LIN {X 0,Y 254.09,Z 840.895,A -85,B 0,C 180,E1 -18628.414,E2 -18628.414} C_VEL
LIN {X 0,Y 254.062,Z 841.128,A -85,B 0,C 180,E1 -18629.999,E2 -18629.999} C_VEL
LIN {X 0,Y 254.089,Z 840.932,A -85,B 0,C 180,E1 -18631.584,E2 -18631.584} C_VEL
LIN {X 0,Y 254.162,Z 840.345,A -85,B 0,C 180,E1 -18633.169,E2 -18633.169} C_VEL
LIN {X 0,Y 254.513,Z 838.113,A -85,B 0,C 180,E1 -18636.232,E2 -18636.232} C_VEL
LIN {X 0,Y 255.051,Z 835.128,A -85,B 0,C 180,E1 -18638.716,E2 -18638.716} C_VEL
LIN {X 0,Y 255.847,Z 831.213,A -85,B 0,C 180,E1 -18641.085,E2 -18641.085} C_VEL
LIN {X 0,Y 257.022,Z 826.141,A -85,B 0,C 180,E1 -18643.438,E2 -18643.438} C_VEL
LIN {X 0,Y 258.473,Z 819.747,A -85,B 0,C 180,E1 -18645.776,E2 -18645.776} C_VEL
LIN {X 0,Y 260.425,Z 811.783,A -85,B 0,C 180,E1 -18648.078,E2 -18648.078} C_VEL
LIN {X 0,Y 262.234,Z 803.648,A -85,B 0,C 180,E1 -18649.976,E2 -18649.976} C_VEL
LIN {X 0,Y 264.141,Z 793.617,A -85,B 0,C 180,E1 -18651.868,E2 -18651.868} C_VEL
LIN {X 0,Y 266.211,Z 782.348,A -85,B 0,C 180,E1 -18653.533,E2 -18653.533} C_VEL
LIN {X 0,Y 267.959,Z 771.245,A -85,B 0,C 180,E1 -18654.81,E2 -18654.81} C_VEL
LIN {X 0,Y 269.52,Z 758.663,A -85,B 0,C 180,E1 -18655.896,E2 -18655.896} C_VEL
LIN {X 0,Y 270.645,Z 746.284,A -85,B 0,C 180,E1 -18656.662,E2 -18656.662} C_VEL
LIN {X 0,Y 271.369,Z 733.669,A -85,B 0,C 180,E1 -18657.157,E2 -18657.157} C_VEL
LIN {X 0,Y 273.583,Z 662.732,A -85,B 0,C 180,E1 -18658.999,E2 -18658.999} C_VEL
LIN {X 0,Y 269.738,Z 639.631,A -85,B 0,C 180,E1 -18660.151,E2 -18660.151} C_VEL
LIN {X 0,Y 267.312,Z 626.531,A -85,B 0,C 180,E1 -18660.876,E2 -18660.876} C_VEL
LIN {X 0,Y 268.617,Z 614.98,A -85,B 0,C 180,E1 -18663.326,E2 -18663.326} C_VEL
LIN {X 0,Y 267.278,Z 607.072,A -85,B 0,C 180,E1 -18665.399,E2 -18665.399} C_VEL
LIN {X 0,Y 264.897,Z 596.537,A -85,B 0,C 180,E1 -18668.397,E2 -18668.397} C_VEL
LIN {X 0,Y 262.253,Z 586.826,A -85,B 0,C 180,E1 -18671.378,E2 -18671.378} C_VEL
LIN {X 0,Y 261.133,Z 583.175,A -85,B 0,C 180,E1 -18672.573,E2 -18672.573} C_VEL
LIN {X 0,Y 265.751,Z 595.35,A -85,B 0,C 180,E1 -18673.336,E2 -18673.336} C_VEL
LIN {X 0,Y 264.419,Z 646.12,A -85,B 0,C 180,E1 -18675.127,E2 -18675.127} C_VEL
LIN {X 0,Y 264.077,Z 660.633,A -85,B 0,C 180,E1 -18675.846,E2 -18675.846} C_VEL
LIN {X 0,Y 263.423,Z 674.387,A -85,B 0,C 180,E1 -18676.869,E2 -18676.869} C_VEL
LIN {X 0,Y 262.637,Z 685.98,A -85,B 0,C 180,E1 -18678.011,E2 -18678.011} C_VEL
LIN {X 0,Y 261.734,Z 697.28,A -85,B 0,C 180,E1 -18679.417,E2 -18679.417} C_VEL
LIN {X 0,Y 260.579,Z 709.014,A -85,B 0,C 180,E1 -18681.254,E2 -18681.254} C_VEL
LIN {X 0,Y 259.619,Z 718.369,A -85,B 0,C 180,E1 -18683.056,E2 -18683.056} C_VEL
LIN {X 0,Y 258.509,Z 722.566,A -85,B 0,C 180,E1 -18683.944,E2 -18683.944} C_VEL
LIN {X 0,Y 255,Z 729.034,A -85,B 0,C 180,E1 -18685.43,E2 -18685.43} C_VEL
LIN {X 0,Y 251.522,Z 734.947,A -85,B 0,C 180,E1 -18687.059,E2 -18687.059} C_VEL
LIN {X 0,Y 250.487,Z 738.277,A -85,B 0,C 180,E1 -18688.153,E2 -18688.153} C_VEL
LIN {X 0,Y 249.964,Z 744.583,A -85,B 0,C 180,E1 -18690.64,E2 -18690.64} C_VEL
LIN {X 0,Y 249.597,Z 749.74,A -85,B 0,C 180,E1 -18693.223,E2 -18693.223} C_VEL
LIN {X 0,Y 249.477,Z 753.747,A -85,B 0,C 180,E1 -18695.89,E2 -18695.89} C_VEL
LIN {X 0,Y 249.746,Z 756.476,A -85,B 0,C 180,E1 -18698.541,E2 -18698.541} C_VEL
LIN {X 0,Y 250.079,Z 757.631,A -85,B 0,C 180,E1 -18700.291,E2 -18700.291} C_VEL
LIN {X 0,Y 250.675,Z 758.421,A -85,B 0,C 180,E1 -18702.401,E2 -18702.401} C_VEL
LIN {X 0,Y 251.933,Z 758.245,A -85,B 0,C 180,E1 -18705.459,E2 -18705.459} C_VEL
LIN {X 0,Y 252.833,Z 757.518,A -85,B 0,C 180,E1 -18707.151,E2 -18707.151} C_VEL
LIN {X 0,Y 253.866,Z 756.267,A -85,B 0,C 180,E1 -18708.826,E2 -18708.826} C_VEL
LIN {X 0,Y 255.812,Z 753.276,A -85,B 0,C 180,E1 -18711.494,E2 -18711.494} C_VEL
LIN {X 0,Y 257.855,Z 749.625,A -85,B 0,C 180,E1 -18713.741,E2 -18713.741} C_VEL
LIN {X 0,Y 260.549,Z 743.915,A -85,B 0,C 180,E1 -18716.368,E2 -18716.368} C_VEL
LIN {X 0,Y 263.546,Z 736.623,A -85,B 0,C 180,E1 -18718.854,E2 -18718.854} C_VEL
LIN {X 0,Y 266.689,Z 727.942,A -85,B 0,C 180,E1 -18721.171,E2 -18721.171} C_VEL
LIN {X 0,Y 269.312,Z 719.321,A -85,B 0,C 180,E1 -18722.992,E2 -18722.992} C_VEL
LIN {X 0,Y 272.249,Z 708.404,A -85,B 0,C 180,E1 -18724.813,E2 -18724.813} C_VEL
LIN {X 0,Y 274.9,Z 696.038,A -85,B 0,C 180,E1 -18726.422,E2 -18726.422} C_VEL
LIN {X 0,Y 276.654,Z 685.777,A -85,B 0,C 180,E1 -18727.481,E2 -18727.481} C_VEL
LIN {X 0,Y 278.215,Z 673.079,A -85,B 0,C 180,E1 -18728.501,E2 -18728.501} C_VEL
LIN {X 0,Y 279.239,Z 659.814,A -85,B 0,C 180,E1 -18729.262,E2 -18729.262} C_VEL
LIN {X 0,Y 281.024,Z 632.819,A -85,B 0,C 180,E1 -18730.403,E2 -18730.403} C_VEL
LIN {X 0,Y 282.345,Z 617.727,A -85,B 0,C 180,E1 -18730.991,E2 -18730.991} C_VEL
LIN {X 0,Y 278.957,Z 610.736,A -85,B 0,C 180,E1 -18732.326,E2 -18732.326} C_VEL
LIN {X 0,Y 274.251,Z 602.926,A -85,B 0,C 180,E1 -18734.285,E2 -18734.285} C_VEL
LIN {X 0,Y 271.133,Z 598.226,A -85,B 0,C 180,E1 -18735.711,E2 -18735.711} C_VEL
LIN {X 0,Y 269.057,Z 595.035,A -85,B 0,C 180,E1 -18736.773,E2 -18736.773} C_VEL
LIN {X 0,Y 266.386,Z 591.181,A -85,B 0,C 180,E1 -18738.242,E2 -18738.242} C_VEL
LIN {X 0,Y 263.756,Z 587.873,A -85,B 0,C 180,E1 -18739.823,E2 -18739.823} C_VEL
LIN {X 0,Y 263.095,Z 586.506,A -85,B 0,C 180,E1 -18740.32,E2 -18740.32} C_VEL
LIN {X 0,Y 260.443,Z 584.072,A -85,B 0,C 180,E1 -18742.197,E2 -18742.197} C_VEL
LIN {X 0,Y 256.402,Z 580.935,A -85,B 0,C 180,E1 -18746.012,E2 -18746.012} C_VEL
LIN {X 0,Y 253.636,Z 580.564,A -85,B 0,C 180,E1 -18750.802,E2 -18750.802} C_VEL
LIN {X 0,Y 253.372,Z 581.196,A -85,B 0,C 180,E1 -18753.694,E2 -18753.694} C_VEL
LIN {X 0,Y 254.251,Z 583.662,A -85,B 0,C 180,E1 -18756.719,E2 -18756.719} C_VEL
LIN {X 0,Y 255.413,Z 586.748,A -85,B 0,C 180,E1 -18759.543,E2 -18759.543} C_VEL
LIN {X 0,Y 258.229,Z 592.704,A -85,B 0,C 180,E1 -18762.875,E2 -18762.875} C_VEL
LIN {X 0,Y 262.198,Z 599.62,A -85,B 0,C 180,E1 -18766.02,E2 -18766.02} C_VEL
LIN {X 0,Y 266.726,Z 608.628,A -85,B 0,C 180,E1 -18768.878,E2 -18768.878} C_VEL
LIN {X 0,Y 270.377,Z 616.548,A -85,B 0,C 180,E1 -18770.836,E2 -18770.836} C_VEL
LIN {X 0,Y 273.12,Z 623.192,A -85,B 0,C 180,E1 -18772.208,E2 -18772.208} C_VEL
LIN {X 0,Y 274.437,Z 626.568,A -85,B 0,C 180,E1 -18772.82,E2 -18772.82} C_VEL
LIN {X 0,Y 276.106,Z 643.037,A -85,B 0,C 180,E1 -18774.364,E2 -18774.364} C_VEL
LIN {X 0,Y 277.294,Z 660.519,A -85,B 0,C 180,E1 -18775.708,E2 -18775.708} C_VEL
LIN {X 0,Y 277.715,Z 677.5,A -85,B 0,C 180,E1 -18776.784,E2 -18776.784} C_VEL
LIN {X 0,Y 277.476,Z 688.854,A -85,B 0,C 180,E1 -18777.368,E2 -18777.368} C_VEL
LIN {X 0,Y 275.097,Z 715.729,A -85,B 0,C 180,E1 -18778.376,E2 -18778.376} C_VEL
LIN {X 0,Y 273.035,Z 729.581,A -85,B 0,C 180,E1 -18779.125,E2 -18779.125} C_VEL
LIN {X 0,Y 270.167,Z 743.428,A -85,B 0,C 180,E1 -18780.167,E2 -18780.167} C_VEL
LIN {X 0,Y 267.203,Z 755.117,A -85,B 0,C 180,E1 -18781.316,E2 -18781.316} C_VEL
LIN {X 0,Y 263.69,Z 767.153,A -85,B 0,C 180,E1 -18782.845,E2 -18782.845} C_VEL
LIN {X 0,Y 262.11,Z 772.187,A -85,B 0,C 180,E1 -18783.583,E2 -18783.583} C_VEL
LIN {X 0,Y 260.479,Z 784.366,A -85,B 0,C 180,E1 -18784.641,E2 -18784.641} C_VEL
LIN {X 0,Y 258.602,Z 795.598,A -85,B 0,C 180,E1 -18785.944,E2 -18785.944} C_VEL
LIN {X 0,Y 256.382,Z 806.998,A -85,B 0,C 180,E1 -18787.647,E2 -18787.647} C_VEL
LIN {X 0,Y 254.432,Z 816.184,A -85,B 0,C 180,E1 -18789.381,E2 -18789.381} C_VEL
LIN {X 0,Y 252.528,Z 825.133,A -85,B 0,C 180,E1 -18791.5,E2 -18791.5} C_VEL
LIN {X 0,Y 250.784,Z 832.715,A -85,B 0,C 180,E1 -18793.727,E2 -18793.727} C_VEL
LIN {X 0,Y 249.202,Z 839.271,A -85,B 0,C 180,E1 -18796.132,E2 -18796.132} C_VEL
LIN {X 0,Y 248.167,Z 844.485,A -85,B 0,C 180,E1 -18798.568,E2 -18798.568} C_VEL
LIN {X 0,Y 247.485,Z 848.517,A -85,B 0,C 180,E1 -18801.016,E2 -18801.016} C_VEL
LIN {X 0,Y 247.074,Z 851.489,A -85,B 0,C 180,E1 -18803.468,E2 -18803.468} C_VEL
LIN {X 0,Y 246.97,Z 852.915,A -85,B 0,C 180,E1 -18805.104,E2 -18805.104} C_VEL
LIN {X 0,Y 246.977,Z 853.923,A -85,B 0,C 180,E1 -18806.739,E2 -18806.739} C_VEL
LIN {X 0,Y 247.025,Z 854.54,A -85,B 0,C 180,E1 -18808.371,E2 -18808.371} C_VEL
LIN {X 0,Y 247.07,Z 854.757,A -85,B 0,C 180,E1 -18810.001,E2 -18810.001} C_VEL
LIN {X 0,Y 247.015,Z 854.529,A -85,B 0,C 180,E1 -18811.632,E2 -18811.632} C_VEL
LIN {X 0,Y 247.011,Z 852.891,A -85,B 0,C 180,E1 -18814.898,E2 -18814.898} C_VEL
LIN {X 0,Y 247.076,Z 851.449,A -85,B 0,C 180,E1 -18816.534,E2 -18816.534} C_VEL
LIN {X 0,Y 247.508,Z 848.465,A -85,B 0,C 180,E1 -18818.986,E2 -18818.986} C_VEL
LIN {X 0,Y 248.152,Z 844.415,A -85,B 0,C 180,E1 -18821.436,E2 -18821.436} C_VEL
LIN {X 0,Y 249.42,Z 838.173,A -85,B 0,C 180,E1 -18824.275,E2 -18824.275} C_VEL
LIN {X 0,Y 251.04,Z 831.372,A -85,B 0,C 180,E1 -18826.677,E2 -18826.677} C_VEL
LIN {X 0,Y 252.834,Z 823.525,A -85,B 0,C 180,E1 -18828.891,E2 -18828.891} C_VEL
LIN {X 0,Y 254.751,Z 814.094,A -85,B 0,C 180,E1 -18831.018,E2 -18831.018} C_VEL
LIN {X 0,Y 256.841,Z 804.471,A -85,B 0,C 180,E1 -18832.738,E2 -18832.738} C_VEL
LIN {X 0,Y 258.885,Z 793.924,A -85,B 0,C 180,E1 -18834.244,E2 -18834.244} C_VEL
LIN {X 0,Y 260.704,Z 782.098,A -85,B 0,C 180,E1 -18835.553,E2 -18835.553} C_VEL
LIN {X 0,Y 262.332,Z 769.822,A -85,B 0,C 180,E1 -18836.557,E2 -18836.557} C_VEL
LIN {X 0,Y 263.569,Z 758.093,A -85,B 0,C 180,E1 -18837.225,E2 -18837.225} C_VEL
LIN {X 0,Y 264.394,Z 743.701,A -85,B 0,C 180,E1 -18837.723,E2 -18837.723} C_VEL
LIN {X 0,Y 266.125,Z 685.702,A -85,B 0,C 180,E1 -18839.262,E2 -18839.262} C_VEL
LIN {X 0,Y 263.423,Z 657.403,A -85,B 0,C 180,E1 -18840.459,E2 -18840.459} C_VEL
LIN {X 0,Y 260.434,Z 634.29,A -85,B 0,C 180,E1 -18841.594,E2 -18841.594} C_VEL
LIN {X 0,Y 259.764,Z 608.016,A -85,B 0,C 180,E1 -18844.496,E2 -18844.496} C_VEL
LIN {X 0,Y 258.866,Z 603.397,A -85,B 0,C 180,E1 -18845.128,E2 -18845.128} C_VEL
LIN {X 0,Y 254.012,Z 587.934,A -85,B 0,C 180,E1 -18847.655,E2 -18847.655} C_VEL
LIN {X 0,Y 251.33,Z 579.796,A -85,B 0,C 180,E1 -18849.096,E2 -18849.096} C_VEL
LIN {X 0,Y 249.033,Z 569.461,A -85,B 0,C 180,E1 -18852.635,E2 -18852.635} C_VEL
LIN {X 0,Y 249.021,Z 569.455,A -85,B 0,C 180,E1 -18857.364,E2 -18857.364} C_VEL
LIN {X 0,Y 249.046,Z 569.45,A -85,B 0,C 180,E1 -18862.201,E2 -18862.201} C_VEL
LIN {X 0,Y 249.046,Z 569.463,A -85,B 0,C 180,E1 -18865.64,E2 -18865.64} C_VEL
LIN {X 0,Y 249.054,Z 569.44,A -85,B 0,C 180,E1 -18869.473,E2 -18869.473} C_VEL
LIN {X 0,Y 249.073,Z 569.452,A -85,B 0,C 180,E1 -18873.162,E2 -18873.162} C_VEL
LIN {X 0,Y 249.064,Z 569.445,A -85,B 0,C 180,E1 -18876.731,E2 -18876.731} C_VEL
LIN {X 0,Y 249.111,Z 569.443,A -85,B 0,C 180,E1 -18880.212,E2 -18880.212} C_VEL
LIN {X 0,Y 249.226,Z 569.419,A -85,B 0,C 180,E1 -18883.621,E2 -18883.621} C_VEL
LIN {X 0,Y 249.247,Z 569.411,A -85,B 0,C 180,E1 -18888.616,E2 -18888.616} C_VEL
LIN {X 0,Y 249.457,Z 569.401,A -85,B 0,C 180,E1 -18891.902,E2 -18891.902} C_VEL
LIN {X 0,Y 249.297,Z 569.419,A -85,B 0,C 180,E1 -18895.149,E2 -18895.149} C_VEL
LIN {X 0,Y 249.677,Z 569.357,A -85,B 0,C 180,E1 -18898.387,E2 -18898.387} C_VEL
LIN {X 0,Y 249.678,Z 569.384,A -85,B 0,C 180,E1 -18901.613,E2 -18901.613} C_VEL
LIN {X 0,Y 249.451,Z 569.391,A -85,B 0,C 180,E1 -18906.729,E2 -18906.729} C_VEL
LIN {X 0,Y 249.392,Z 569.415,A -85,B 0,C 180,E1 -18909.735,E2 -18909.735} C_VEL
LIN {X 0,Y 249.204,Z 569.436,A -85,B 0,C 180,E1 -18914.704,E2 -18914.704} C_VEL
LIN {X 0,Y 249.142,Z 569.432,A -85,B 0,C 180,E1 -18918.077,E2 -18918.077} C_VEL
LIN {X 0,Y 249.09,Z 569.453,A -85,B 0,C 180,E1 -18921.518,E2 -18921.518} C_VEL
LIN {X 0,Y 249.133,Z 569.43,A -85,B 0,C 180,E1 -18925.482,E2 -18925.482} C_VEL
LIN {X 0,Y 249.086,Z 569.455,A -85,B 0,C 180,E1 -18928.993,E2 -18928.993} C_VEL
LIN {X 0,Y 249.033,Z 569.46,A -85,B 0,C 180,E1 -18932.426,E2 -18932.426} C_VEL
LIN {X 0,Y 249.059,Z 569.453,A -85,B 0,C 180,E1 -18936.341,E2 -18936.341} C_VEL
LIN {X 0,Y 249.029,Z 569.46,A -85,B 0,C 180,E1 -18940.474,E2 -18940.474} C_VEL
LIN {X 0,Y 249.011,Z 569.51,A -85,B 0,C 180,E1 -18943.137,E2 -18943.137} C_VEL
LIN {X 0,Y 253.699,Z 582.025,A -85,B 0,C 180,E1 -18947.232,E2 -18947.232} C_VEL
LIN {X 0,Y 257.124,Z 592.661,A -85,B 0,C 180,E1 -18950.444,E2 -18950.444} C_VEL
LIN {X 0,Y 260.154,Z 603.871,A -85,B 0,C 180,E1 -18953.535,E2 -18953.535} C_VEL
LIN {X 0,Y 262.882,Z 616.414,A -85,B 0,C 180,E1 -18956.711,E2 -18956.711} C_VEL
LIN {X 0,Y 262.799,Z 619.429,A -85,B 0,C 180,E1 -18957.335,E2 -18957.335} C_VEL
LIN {X 0,Y 262.047,Z 625.84,A -85,B 0,C 180,E1 -18958.543,E2 -18958.543} C_VEL
LIN {X 0,Y 266.616,Z 654.96,A -85,B 0,C 180,E1 -18960.056,E2 -18960.056} C_VEL
LIN {X 0,Y 267.466,Z 661.868,A -85,B 0,C 180,E1 -18960.372,E2 -18960.372} C_VEL
LIN {X 0,Y 264.785,Z 738.66,A -85,B 0,C 180,E1 -18962.429,E2 -18962.429} C_VEL
LIN {X 0,Y 263.808,Z 751.811,A -85,B 0,C 180,E1 -18963.07,E2 -18963.07} C_VEL
LIN {X 0,Y 262.417,Z 764.297,A -85,B 0,C 180,E1 -18963.988,E2 -18963.988} C_VEL
LIN {X 0,Y 260.839,Z 775.507,A -85,B 0,C 180,E1 -18965.101,E2 -18965.101} C_VEL
LIN {X 0,Y 258.758,Z 787.098,A -85,B 0,C 180,E1 -18966.594,E2 -18966.594} C_VEL
LIN {X 0,Y 256.708,Z 797.852,A -85,B 0,C 180,E1 -18968.393,E2 -18968.393} C_VEL
LIN {X 0,Y 254.893,Z 806.829,A -85,B 0,C 180,E1 -18970.273,E2 -18970.273} C_VEL
LIN {X 0,Y 252.71,Z 815.756,A -85,B 0,C 180,E1 -18972.604,E2 -18972.604} C_VEL
LIN {X 0,Y 250.925,Z 822.969,A -85,B 0,C 180,E1 -18974.984,E2 -18974.984} C_VEL
LIN {X 0,Y 249.294,Z 829.586,A -85,B 0,C 180,E1 -18977.792,E2 -18977.792} C_VEL
LIN {X 0,Y 248.31,Z 833.924,A -85,B 0,C 180,E1 -18980.221,E2 -18980.221} C_VEL
LIN {X 0,Y 247.845,Z 836.205,A -85,B 0,C 180,E1 -18981.848,E2 -18981.848} C_VEL
LIN {X 0,Y 247.389,Z 838.457,A -85,B 0,C 180,E1 -18983.885,E2 -18983.885} C_VEL
LIN {X 0,Y 247.087,Z 840.476,A -85,B 0,C 180,E1 -18986.738,E2 -18986.738} C_VEL
LIN {X 0,Y 246.992,Z 841.32,A -85,B 0,C 180,E1 -18989.999,E2 -18989.999} C_VEL
LIN {X 0,Y 247,Z 841.125,A -85,B 0,C 180,E1 -18991.629,E2 -18991.629} C_VEL
LIN {X 0,Y 247.084,Z 840.537,A -85,B 0,C 180,E1 -18993.26,E2 -18993.26} C_VEL
LIN {X 0,Y 247.418,Z 838.511,A -85,B 0,C 180,E1 -18996.177,E2 -18996.177} C_VEL
LIN {X 0,Y 248.042,Z 835.319,A -85,B 0,C 180,E1 -18998.964,E2 -18998.964} C_VEL
LIN {X 0,Y 248.875,Z 831.404,A -85,B 0,C 180,E1 -19001.399,E2 -19001.399} C_VEL
LIN {X 0,Y 250.114,Z 826.331,A -85,B 0,C 180,E1 -19003.817,E2 -19003.817} C_VEL
LIN {X 0,Y 251.642,Z 819.935,A -85,B 0,C 180,E1 -19006.216,E2 -19006.216} C_VEL
LIN {X 0,Y 253.691,Z 811.969,A -85,B 0,C 180,E1 -19008.576,E2 -19008.576} C_VEL
LIN {X 0,Y 255.675,Z 803.234,A -85,B 0,C 180,E1 -19010.653,E2 -19010.653} C_VEL
LIN {X 0,Y 257.574,Z 793.796,A -85,B 0,C 180,E1 -19012.456,E2 -19012.456} C_VEL
LIN {X 0,Y 259.738,Z 782.522,A -85,B 0,C 180,E1 -19014.156,E2 -19014.156} C_VEL
LIN {X 0,Y 261.545,Z 771.411,A -85,B 0,C 180,E1 -19015.462,E2 -19015.462} C_VEL
LIN {X 0,Y 263.034,Z 760.044,A -85,B 0,C 180,E1 -19016.477,E2 -19016.477} C_VEL
LIN {X 0,Y 264.257,Z 747.263,A -85,B 0,C 180,E1 -19017.306,E2 -19017.306} C_VEL
LIN {X 0,Y 265.04,Z 735.241,A -85,B 0,C 180,E1 -19017.807,E2 -19017.807} C_VEL
LIN {X 0,Y 267.411,Z 663.775,A -85,B 0,C 180,E1 -19019.704,E2 -19019.704} C_VEL
LIN {X 0,Y 263.005,Z 637.473,A -85,B 0,C 180,E1 -19021.076,E2 -19021.076} C_VEL
LIN {X 0,Y 261,Z 626.634,A -85,B 0,C 180,E1 -19021.701,E2 -19021.701} C_VEL
LIN {X 0,Y 262.114,Z 617.018,A -85,B 0,C 180,E1 -19023.778,E2 -19023.778} C_VEL
LIN {X 0,Y 260.389,Z 607.236,A -85,B 0,C 180,E1 -19026.424,E2 -19026.424} C_VEL
LIN {X 0,Y 257.403,Z 594.767,A -85,B 0,C 180,E1 -19030.137,E2 -19030.137} C_VEL
LIN {X 0,Y 255.388,Z 587.888,A -85,B 0,C 180,E1 -19032.362,E2 -19032.362} C_VEL
LIN {X 0,Y 256.803,Z 590.995,A -85,B 0,C 180,E1 -19032.577,E2 -19032.577} C_VEL
LIN {X 0,Y 259.068,Z 597.539,A -85,B 0,C 180,E1 -19032.98,E2 -19032.98} C_VEL
LIN {X 0,Y 257.655,Z 639.19,A -85,B 0,C 180,E1 -19034.476,E2 -19034.476} C_VEL
LIN {X 0,Y 257.372,Z 656.39,A -85,B 0,C 180,E1 -19035.21,E2 -19035.21} C_VEL
LIN {X 0,Y 256.764,Z 670.302,A -85,B 0,C 180,E1 -19036.144,E2 -19036.144} C_VEL
LIN {X 0,Y 256.037,Z 682.338,A -85,B 0,C 180,E1 -19037.244,E2 -19037.244} C_VEL
LIN {X 0,Y 255.137,Z 694.009,A -85,B 0,C 180,E1 -19038.616,E2 -19038.616} C_VEL
LIN {X 0,Y 253.941,Z 706.445,A -85,B 0,C 180,E1 -19040.465,E2 -19040.465} C_VEL
LIN {X 0,Y 252.919,Z 716.407,A -85,B 0,C 180,E1 -19042.314,E2 -19042.314} C_VEL
LIN {X 0,Y 251.822,Z 726.426,A -85,B 0,C 180,E1 -19044.612,E2 -19044.612} C_VEL
LIN {X 0,Y 250.987,Z 733.793,A -85,B 0,C 180,E1 -19046.675,E2 -19046.675} C_VEL
LIN {X 0,Y 250.487,Z 738.277,A -85,B 0,C 180,E1 -19048.153,E2 -19048.153} C_VEL
LIN {X 0,Y 249.499,Z 741.431,A -85,B 0,C 180,E1 -19049.279,E2 -19049.279} C_VEL
LIN {X 0,Y 246.27,Z 746.193,A -85,B 0,C 180,E1 -19051.148,E2 -19051.148} C_VEL
LIN {X 0,Y 243.18,Z 750.314,A -85,B 0,C 180,E1 -19053.139,E2 -19053.139} C_VEL
LIN {X 0,Y 242.435,Z 752.446,A -85,B 0,C 180,E1 -19054.432,E2 -19054.432} C_VEL
LIN {X 0,Y 242.422,Z 754.701,A -85,B 0,C 180,E1 -19056.054,E2 -19056.054} C_VEL
LIN {X 0,Y 242.601,Z 756.771,A -85,B 0,C 180,E1 -19057.969,E2 -19057.969} C_VEL
LIN {X 0,Y 242.91,Z 758.159,A -85,B 0,C 180,E1 -19059.684,E2 -19059.684} C_VEL
LIN {X 0,Y 243.577,Z 759.382,A -85,B 0,C 180,E1 -19062.198,E2 -19062.198} C_VEL
LIN {X 0,Y 244.686,Z 759.623,A -85,B 0,C 180,E1 -19065.019,E2 -19065.019} C_VEL
LIN {X 0,Y 245.597,Z 759.147,A -85,B 0,C 180,E1 -19066.766,E2 -19066.766} C_VEL
LIN {X 0,Y 246.642,Z 758.193,A -85,B 0,C 180,E1 -19068.494,E2 -19068.494} C_VEL
LIN {X 0,Y 248.753,Z 755.486,A -85,B 0,C 180,E1 -19071.422,E2 -19071.422} C_VEL
LIN {X 0,Y 250.65,Z 752.454,A -85,B 0,C 180,E1 -19073.56,E2 -19073.56} C_VEL
LIN {X 0,Y 253.518,Z 747.121,A -85,B 0,C 180,E1 -19076.329,E2 -19076.329} C_VEL
LIN {X 0,Y 256.507,Z 740.69,A -85,B 0,C 180,E1 -19078.822,E2 -19078.822} C_VEL
LIN {X 0,Y 259.282,Z 733.984,A -85,B 0,C 180,E1 -19080.854,E2 -19080.854} C_VEL
LIN {X 0,Y 262.174,Z 725.886,A -85,B 0,C 180,E1 -19082.839,E2 -19082.839} C_VEL
LIN {X 0,Y 265.177,Z 716.123,A -85,B 0,C 180,E1 -19084.751,E2 -19084.751} C_VEL
LIN {X 0,Y 268.104,Z 705.231,A -85,B 0,C 180,E1 -19086.434,E2 -19086.434} C_VEL
LIN {X 0,Y 270.598,Z 693.198,A -85,B 0,C 180,E1 -19087.894,E2 -19087.894} C_VEL
LIN {X 0,Y 272.646,Z 680.632,A -85,B 0,C 180,E1 -19089.053,E2 -19089.053} C_VEL
LIN {X 0,Y 274.025,Z 667.183,A -85,B 0,C 180,E1 -19089.999,E2 -19089.999} C_VEL
LIN {X 0,Y 275.305,Z 648.329,A -85,B 0,C 180,E1 -19090.905,E2 -19090.905} C_VEL
LIN {X 0,Y 277.684,Z 620.883,A -85,B 0,C 180,E1 -19092.021,E2 -19092.021} C_VEL
LIN {X 0,Y 275.405,Z 615.981,A -85,B 0,C 180,E1 -19092.991,E2 -19092.991} C_VEL
LIN {X 0,Y 270.894,Z 608.299,A -85,B 0,C 180,E1 -19094.985,E2 -19094.985} C_VEL
LIN {X 0,Y 266.537,Z 601.354,A -85,B 0,C 180,E1 -19097.216,E2 -19097.216} C_VEL
LIN {X 0,Y 263.964,Z 597.532,A -85,B 0,C 180,E1 -19098.733,E2 -19098.733} C_VEL
LIN {X 0,Y 261.41,Z 594.02,A -85,B 0,C 180,E1 -19100.39,E2 -19100.39} C_VEL
LIN {X 0,Y 260.837,Z 593.011,A -85,B 0,C 180,E1 -19100.839,E2 -19100.839} C_VEL
LIN {X 0,Y 258.203,Z 590.417,A -85,B 0,C 180,E1 -19102.822,E2 -19102.822} C_VEL
LIN {X 0,Y 255.21,Z 588.146,A -85,B 0,C 180,E1 -19105.729,E2 -19105.729} C_VEL
LIN {X 0,Y 253.396,Z 587.616,A -85,B 0,C 180,E1 -19108.132,E2 -19108.132} C_VEL
LIN {X 0,Y 252.16,Z 587.56,A -85,B 0,C 180,E1 -19111.129,E2 -19111.129} C_VEL
LIN {X 0,Y 251.929,Z 588.384,A -85,B 0,C 180,E1 -19113.913,E2 -19113.913} C_VEL
LIN {X 0,Y 252.608,Z 590.937,A -85,B 0,C 180,E1 -19116.996,E2 -19116.996} C_VEL
LIN {X 0,Y 253.732,Z 593.511,A -85,B 0,C 180,E1 -19119.214,E2 -19119.214} C_VEL
LIN {X 0,Y 256.46,Z 599.656,A -85,B 0,C 180,E1 -19122.636,E2 -19122.636} C_VEL
LIN {X 0,Y 259.717,Z 605.662,A -85,B 0,C 180,E1 -19125.384,E2 -19125.384} C_VEL
LIN {X 0,Y 263.844,Z 614.341,A -85,B 0,C 180,E1 -19128.195,E2 -19128.195} C_VEL
LIN {X 0,Y 267.113,Z 621.867,A -85,B 0,C 180,E1 -19130.108,E2 -19130.108} C_VEL
LIN {X 0,Y 269.665,Z 628.359,A -85,B 0,C 180,E1 -19131.477,E2 -19131.477} C_VEL
LIN {X 0,Y 270.426,Z 630.865,A -85,B 0,C 180,E1 -19131.914,E2 -19131.914} C_VEL
LIN {X 0,Y 271.947,Z 648.046,A -85,B 0,C 180,E1 -19133.533,E2 -19133.533} C_VEL
LIN {X 0,Y 272.788,Z 665.923,A -85,B 0,C 180,E1 -19134.925,E2 -19134.925} C_VEL
LIN {X 0,Y 272.877,Z 684.026,A -85,B 0,C 180,E1 -19136.018,E2 -19136.018} C_VEL
LIN {X 0,Y 272.525,Z 691.059,A -85,B 0,C 180,E1 -19136.346,E2 -19136.346} C_VEL
LIN {X 0,Y 270.201,Z 714.937,A -85,B 0,C 180,E1 -19137.283,E2 -19137.283} C_VEL
LIN {X 0,Y 268.004,Z 728.536,A -85,B 0,C 180,E1 -19138.038,E2 -19138.038} C_VEL
LIN {X 0,Y 265,Z 742.273,A -85,B 0,C 180,E1 -19139.082,E2 -19139.082} C_VEL
LIN {X 0,Y 261.917,Z 753.948,A -85,B 0,C 180,E1 -19140.239,E2 -19140.239} C_VEL
LIN {X 0,Y 258.233,Z 765.958,A -85,B 0,C 180,E1 -19141.781,E2 -19141.781} C_VEL
LIN {X 0,Y 255.527,Z 773.89,A -85,B 0,C 180,E1 -19143.013,E2 -19143.013} C_VEL
LIN {X 0,Y 253.804,Z 785.941,A -85,B 0,C 180,E1 -19144.145,E2 -19144.145} C_VEL
LIN {X 0,Y 251.864,Z 796.83,A -85,B 0,C 180,E1 -19145.478,E2 -19145.478} C_VEL
LIN {X 0,Y 249.568,Z 807.936,A -85,B 0,C 180,E1 -19147.221,E2 -19147.221} C_VEL
LIN {X 0,Y 247.366,Z 817.776,A -85,B 0,C 180,E1 -19149.2,E2 -19149.2} C_VEL
LIN {X 0,Y 245.619,Z 825.59,A -85,B 0,C 180,E1 -19151.149,E2 -19151.149} C_VEL
LIN {X 0,Y 243.665,Z 833.749,A -85,B 0,C 180,E1 -19153.669,E2 -19153.669} C_VEL
LIN {X 0,Y 242.287,Z 839.081,A -85,B 0,C 180,E1 -19155.728,E2 -19155.728} C_VEL
LIN {X 0,Y 241.187,Z 844.293,A -85,B 0,C 180,E1 -19158.232,E2 -19158.232} C_VEL
LIN {X 0,Y 240.44,Z 848.325,A -85,B 0,C 180,E1 -19160.75,E2 -19160.75} C_VEL
LIN {X 0,Y 239.997,Z 851.296,A -85,B 0,C 180,E1 -19163.275,E2 -19163.275} C_VEL
LIN {X 0,Y 239.88,Z 852.722,A -85,B 0,C 180,E1 -19164.959,E2 -19164.959} C_VEL
LIN {X 0,Y 239.877,Z 853.73,A -85,B 0,C 180,E1 -19166.642,E2 -19166.642} C_VEL
LIN {X 0,Y 239.931,Z 854.347,A -85,B 0,C 180,E1 -19168.323,E2 -19168.323} C_VEL
LIN {X 0,Y 239.997,Z 854.565,A -85,B 0,C 180,E1 -19170.001,E2 -19170.001} C_VEL
LIN {X 0,Y 239.922,Z 854.336,A -85,B 0,C 180,E1 -19171.68,E2 -19171.68} C_VEL
LIN {X 0,Y 239.921,Z 852.697,A -85,B 0,C 180,E1 -19175.043,E2 -19175.043} C_VEL
LIN {X 0,Y 240.001,Z 851.255,A -85,B 0,C 180,E1 -19176.728,E2 -19176.728} C_VEL
LIN {X 0,Y 240.456,Z 848.27,A -85,B 0,C 180,E1 -19179.252,E2 -19179.252} C_VEL
LIN {X 0,Y 241.166,Z 844.221,A -85,B 0,C 180,E1 -19181.772,E2 -19181.772} C_VEL
LIN {X 0,Y 242.529,Z 837.98,A -85,B 0,C 180,E1 -19184.689,E2 -19184.689} C_VEL
LIN {X 0,Y 244.182,Z 831.178,A -85,B 0,C 180,E1 -19187.16,E2 -19187.16} C_VEL
LIN {X 0,Y 245.941,Z 824.007,A -85,B 0,C 180,E1 -19189.252,E2 -19189.252} C_VEL
LIN {X 0,Y 247.699,Z 815.836,A -85,B 0,C 180,E1 -19191.209,E2 -19191.209} C_VEL
LIN {X 0,Y 250.035,Z 805.446,A -85,B 0,C 180,E1 -19193.174,E2 -19193.174} C_VEL
LIN {X 0,Y 252.129,Z 795.159,A -85,B 0,C 180,E1 -19194.717,E2 -19194.717} C_VEL
LIN {X 0,Y 254.048,Z 783.861,A -85,B 0,C 180,E1 -19196.052,E2 -19196.052} C_VEL
LIN {X 0,Y 255.847,Z 770.923,A -85,B 0,C 180,E1 -19197.174,E2 -19197.174} C_VEL
LIN {X 0,Y 257.188,Z 758.88,A -85,B 0,C 180,E1 -19197.9,E2 -19197.9} C_VEL
LIN {X 0,Y 258.06,Z 745.717,A -85,B 0,C 180,E1 -19198.396,E2 -19198.396} C_VEL
LIN {X 0,Y 259.901,Z 685.945,A -85,B 0,C 180,E1 -19200.023,E2 -19200.023} C_VEL
LIN {X 0,Y 257.251,Z 657.764,A -85,B 0,C 180,E1 -19201.257,E2 -19201.257} C_VEL
LIN {X 0,Y 254.175,Z 634.196,A -85,B 0,C 180,E1 -19202.469,E2 -19202.469} C_VEL
LIN {X 0,Y 253.843,Z 610.077,A -85,B 0,C 180,E1 -19205.241,E2 -19205.241} C_VEL
LIN {X 0,Y 252.81,Z 605.724,A -85,B 0,C 180,E1 -19205.882,E2 -19205.882} C_VEL
LIN {X 0,Y 249.822,Z 596.027,A -85,B 0,C 180,E1 -19207.512,E2 -19207.512} C_VEL
LIN {X 0,Y 245.651,Z 582.707,A -85,B 0,C 180,E1 -19209.925,E2 -19209.925} C_VEL
LIN {X 0,Y 242.755,Z 573.824,A -85,B 0,C 180,E1 -19211.75,E2 -19211.75} C_VEL
LIN {X 0,Y 241.964,Z 570.336,A -85,B 0,C 180,E1 -19213.076,E2 -19213.076} C_VEL
LIN {X 0,Y 241.939,Z 570.346,A -85,B 0,C 180,E1 -19216.571,E2 -19216.571} C_VEL
LIN {X 0,Y 241.959,Z 570.345,A -85,B 0,C 180,E1 -19220.281,E2 -19220.281} C_VEL
LIN {X 0,Y 241.983,Z 570.329,A -85,B 0,C 180,E1 -19224.488,E2 -19224.488} C_VEL
LIN {X 0,Y 241.977,Z 570.321,A -85,B 0,C 180,E1 -19228.48,E2 -19228.48} C_VEL
LIN {X 0,Y 242.01,Z 570.339,A -85,B 0,C 180,E1 -19232.313,E2 -19232.313} C_VEL
LIN {X 0,Y 242.044,Z 570.311,A -85,B 0,C 180,E1 -19236.015,E2 -19236.015} C_VEL
LIN {X 0,Y 242.038,Z 570.331,A -85,B 0,C 180,E1 -19239.608,E2 -19239.608} C_VEL
LIN {X 0,Y 242.166,Z 570.294,A -85,B 0,C 180,E1 -19243.278,E2 -19243.278} C_VEL
LIN {X 0,Y 242.183,Z 570.294,A -85,B 0,C 180,E1 -19248.28,E2 -19248.28} C_VEL
LIN {X 0,Y 242.403,Z 570.276,A -85,B 0,C 180,E1 -19251.665,E2 -19251.665} C_VEL
LIN {X 0,Y 242.258,Z 570.297,A -85,B 0,C 180,E1 -19255.007,E2 -19255.007} C_VEL
LIN {X 0,Y 242.638,Z 570.232,A -85,B 0,C 180,E1 -19258.34,E2 -19258.34} C_VEL
LIN {X 0,Y 242.638,Z 570.261,A -85,B 0,C 180,E1 -19261.66,E2 -19261.66} C_VEL
LIN {X 0,Y 242.431,Z 570.266,A -85,B 0,C 180,E1 -19266.706,E2 -19266.706} C_VEL
LIN {X 0,Y 242.317,Z 570.294,A -85,B 0,C 180,E1 -19270.022,E2 -19270.022} C_VEL
LIN {X 0,Y 242.167,Z 570.317,A -85,B 0,C 180,E1 -19275.141,E2 -19275.141} C_VEL
LIN {X 0,Y 242.075,Z 570.307,A -85,B 0,C 180,E1 -19278.624,E2 -19278.624} C_VEL
LIN {X 0,Y 242.016,Z 570.34,A -85,B 0,C 180,E1 -19282.18,E2 -19282.18} C_VEL
LIN {X 0,Y 242.07,Z 570.311,A -85,B 0,C 180,E1 -19285.838,E2 -19285.838} C_VEL
LIN {X 0,Y 242.033,Z 570.325,A -85,B 0,C 180,E1 -19289.58,E2 -19289.58} C_VEL
LIN {X 0,Y 241.985,Z 570.346,A -85,B 0,C 180,E1 -19293.492,E2 -19293.492} C_VEL
LIN {X 0,Y 242.002,Z 570.345,A -85,B 0,C 180,E1 -19297.58,E2 -19297.58} C_VEL
LIN {X 0,Y 241.943,Z 570.406,A -85,B 0,C 180,E1 -19301.714,E2 -19301.714} C_VEL
LIN {X 0,Y 246.074,Z 581.311,A -85,B 0,C 180,E1 -19305.563,E2 -19305.563} C_VEL
LIN {X 0,Y 249.569,Z 591.221,A -85,B 0,C 180,E1 -19308.705,E2 -19308.705} C_VEL
LIN {X 0,Y 252.451,Z 601.155,A -85,B 0,C 180,E1 -19311.643,E2 -19311.643} C_VEL
LIN {X 0,Y 255.514,Z 614.014,A -85,B 0,C 180,E1 -19315.069,E2 -19315.069} C_VEL
LIN {X 0,Y 256.572,Z 619.642,A -85,B 0,C 180,E1 -19316.465,E2 -19316.465} C_VEL
LIN {X 0,Y 255.815,Z 626,A -85,B 0,C 180,E1 -19317.697,E2 -19317.697} C_VEL
LIN {X 0,Y 260.073,Z 653.291,A -85,B 0,C 180,E1 -19319.166,E2 -19319.166} C_VEL
LIN {X 0,Y 261.288,Z 663.431,A -85,B 0,C 180,E1 -19319.645,E2 -19319.645} C_VEL
LIN {X 0,Y 258.529,Z 738.791,A -85,B 0,C 180,E1 -19321.703,E2 -19321.703} C_VEL
LIN {X 0,Y 257.518,Z 751.975,A -85,B 0,C 180,E1 -19322.357,E2 -19322.357} C_VEL
LIN {X 0,Y 256.073,Z 764.47,A -85,B 0,C 180,E1 -19323.293,E2 -19323.293} C_VEL
LIN {X 0,Y 254.434,Z 775.687,A -85,B 0,C 180,E1 -19324.43,E2 -19324.43} C_VEL
LIN {X 0,Y 252.256,Z 787.284,A -85,B 0,C 180,E1 -19325.954,E2 -19325.954} C_VEL
LIN {X 0,Y 250.111,Z 798.041,A -85,B 0,C 180,E1 -19327.793,E2 -19327.793} C_VEL
LIN {X 0,Y 248.187,Z 807.16,A -85,B 0,C 180,E1 -19329.752,E2 -19329.752} C_VEL
LIN {X 0,Y 245.954,Z 815.947,A -85,B 0,C 180,E1 -19332.11,E2 -19332.11} C_VEL
LIN {X 0,Y 244.07,Z 823.162,A -85,B 0,C 180,E1 -19334.551,E2 -19334.551} C_VEL
LIN {X 0,Y 242.342,Z 829.78,A -85,B 0,C 180,E1 -19337.436,E2 -19337.436} C_VEL
LIN {X 0,Y 241.304,Z 834.118,A -85,B 0,C 180,E1 -19339.935,E2 -19339.935} C_VEL
LIN {X 0,Y 240.807,Z 836.398,A -85,B 0,C 180,E1 -19341.608,E2 -19341.608} C_VEL
LIN {X 0,Y 240.304,Z 838.834,A -85,B 0,C 180,E1 -19343.923,E2 -19343.923} C_VEL
LIN {X 0,Y 240.01,Z 840.669,A -85,B 0,C 180,E1 -19346.641,E2 -19346.641} C_VEL
LIN {X 0,Y 239.923,Z 841.512,A -85,B 0,C 180,E1 -19349.999,E2 -19349.999} C_VEL
LIN {X 0,Y 239.912,Z 841.317,A -85,B 0,C 180,E1 -19351.677,E2 -19351.677} C_VEL
LIN {X 0,Y 240.008,Z 840.729,A -85,B 0,C 180,E1 -19353.356,E2 -19353.356} C_VEL
LIN {X 0,Y 240.318,Z 838.914,A -85,B 0,C 180,E1 -19356.109,E2 -19356.109} C_VEL
LIN {X 0,Y 241.011,Z 835.511,A -85,B 0,C 180,E1 -19359.228,E2 -19359.228} C_VEL
LIN {X 0,Y 241.916,Z 831.595,A -85,B 0,C 180,E1 -19361.732,E2 -19361.732} C_VEL
LIN {X 0,Y 243.219,Z 826.52,A -85,B 0,C 180,E1 -19364.216,E2 -19364.216} C_VEL
LIN {X 0,Y 244.83,Z 820.123,A -85,B 0,C 180,E1 -19366.68,E2 -19366.68} C_VEL
LIN {X 0,Y 246.979,Z 812.154,A -85,B 0,C 180,E1 -19369.1,E2 -19369.1} C_VEL
LIN {X 0,Y 248.908,Z 803.975,A -85,B 0,C 180,E1 -19371.106,E2 -19371.106} C_VEL
LIN {X 0,Y 251.034,Z 793.976,A -85,B 0,C 180,E1 -19373.074,E2 -19373.074} C_VEL
LIN {X 0,Y 253.288,Z 782.696,A -85,B 0,C 180,E1 -19374.812,E2 -19374.812} C_VEL
LIN {X 0,Y 255.161,Z 771.578,A -85,B 0,C 180,E1 -19376.146,E2 -19376.146} C_VEL
LIN {X 0,Y 256.843,Z 758.97,A -85,B 0,C 180,E1 -19377.277,E2 -19377.277} C_VEL
LIN {X 0,Y 258.069,Z 746.551,A -85,B 0,C 180,E1 -19378.073,E2 -19378.073} C_VEL
LIN {X 0,Y 258.862,Z 733.81,A -85,B 0,C 180,E1 -19378.586,E2 -19378.586} C_VEL
LIN {X 0,Y 261.202,Z 664.421,A -85,B 0,C 180,E1 -19380.466,E2 -19380.466} C_VEL
LIN {X 0,Y 256.549,Z 636.372,A -85,B 0,C 180,E1 -19381.987,E2 -19381.987} C_VEL
LIN {X 0,Y 254.753,Z 626.786,A -85,B 0,C 180,E1 -19382.579,E2 -19382.579} C_VEL
LIN {X 0,Y 255.597,Z 618.433,A -85,B 0,C 180,E1 -19384.422,E2 -19384.422} C_VEL
LIN {X 0,Y 253.4,Z 607.174,A -85,B 0,C 180,E1 -19387.599,E2 -19387.599} C_VEL
LIN {X 0,Y 250.842,Z 596.665,A -85,B 0,C 180,E1 -19390.845,E2 -19390.845} C_VEL
LIN {X 0,Y 249.715,Z 592.683,A -85,B 0,C 180,E1 -19392.171,E2 -19392.171} C_VEL
LIN {X 0,Y 251.194,Z 595.873,A -85,B 0,C 180,E1 -19392.398,E2 -19392.398} C_VEL
LIN {X 0,Y 252.164,Z 599.245,A -85,B 0,C 180,E1 -19392.596,E2 -19392.596} C_VEL
LIN {X 0,Y 250.725,Z 641.596,A -85,B 0,C 180,E1 -19394.176,E2 -19394.176} C_VEL
LIN {X 0,Y 250.442,Z 657.573,A -85,B 0,C 180,E1 -19394.891,E2 -19394.891} C_VEL
LIN {X 0,Y 249.858,Z 670.554,A -85,B 0,C 180,E1 -19395.781,E2 -19395.781} C_VEL
LIN {X 0,Y 249.055,Z 683.719,A -85,B 0,C 180,E1 -19397.011,E2 -19397.011} C_VEL
LIN {X 0,Y 248.015,Z 696.014,A -85,B 0,C 180,E1 -19398.518,E2 -19398.518} C_VEL
LIN {X 0,Y 246.972,Z 706.977,A -85,B 0,C 180,E1 -19400.201,E2 -19400.201} C_VEL
LIN {X 0,Y 245.901,Z 716.993,A -85,B 0,C 180,E1 -19402.085,E2 -19402.085} C_VEL
LIN {X 0,Y 244.795,Z 727.117,A -85,B 0,C 180,E1 -19404.453,E2 -19404.453} C_VEL
LIN {X 0,Y 243.817,Z 735.271,A -85,B 0,C 180,E1 -19406.792,E2 -19406.792} C_VEL
LIN {X 0,Y 243.123,Z 742.781,A -85,B 0,C 180,E1 -19409.505,E2 -19409.505} C_VEL
LIN {X 0,Y 242.633,Z 749.017,A -85,B 0,C 180,E1 -19412.39,E2 -19412.39} C_VEL
LIN {X 0,Y 242.435,Z 752.446,A -85,B 0,C 180,E1 -19414.432,E2 -19414.432} C_VEL
LIN {X 0,Y 241.758,Z 754.381,A -85,B 0,C 180,E1 -19415.746,E2 -19415.746} C_VEL
LIN {X 0,Y 239.078,Z 757.134,A -85,B 0,C 180,E1 -19417.924,E2 -19417.924} C_VEL
LIN {X 0,Y 236.985,Z 758.9,A -85,B 0,C 180,E1 -19419.724,E2 -19419.724} C_VEL
LIN {X 0,Y 236.298,Z 759.884,A -85,B 0,C 180,E1 -19421.13,E2 -19421.13} C_VEL
LIN {X 0,Y 236.352,Z 760.115,A -85,B 0,C 180,E1 -19421.604,E2 -19421.604} C_VEL
LIN {X 0,Y 237.445,Z 760.847,A -85,B 0,C 180,E1 -19424.55,E2 -19424.55} C_VEL
LIN {X 0,Y 238.446,Z 760.579,A -85,B 0,C 180,E1 -19426.559,E2 -19426.559} C_VEL
LIN {X 0,Y 239.393,Z 759.977,A -85,B 0,C 180,E1 -19428.141,E2 -19428.141} C_VEL
LIN {X 0,Y 240.577,Z 758.849,A -85,B 0,C 180,E1 -19429.905,E2 -19429.905} C_VEL
LIN {X 0,Y 242.64,Z 756.242,A -85,B 0,C 180,E1 -19432.511,E2 -19432.511} C_VEL
LIN {X 0,Y 245.141,Z 752.486,A -85,B 0,C 180,E1 -19435.066,E2 -19435.066} C_VEL
LIN {X 0,Y 247.898,Z 747.526,A -85,B 0,C 180,E1 -19437.563,E2 -19437.563} C_VEL
LIN {X 0,Y 251.062,Z 741.134,A -85,B 0,C 180,E1 -19440,E2 -19440} C_VEL
LIN {X 0,Y 254.423,Z 733.327,A -85,B 0,C 180,E1 -19442.314,E2 -19442.314} C_VEL
LIN {X 0,Y 257.461,Z 724.991,A -85,B 0,C 180,E1 -19444.305,E2 -19444.305} C_VEL
LIN {X 0,Y 260.396,Z 716.03,A -85,B 0,C 180,E1 -19446.003,E2 -19446.003} C_VEL
LIN {X 0,Y 262.921,Z 706.924,A -85,B 0,C 180,E1 -19447.411,E2 -19447.411} C_VEL
LIN {X 0,Y 265.555,Z 695.346,A -85,B 0,C 180,E1 -19448.864,E2 -19448.864} C_VEL
LIN {X 0,Y 267.69,Z 683.478,A -85,B 0,C 180,E1 -19450.017,E2 -19450.017} C_VEL
LIN {X 0,Y 269.245,Z 670.621,A -85,B 0,C 180,E1 -19450.973,E2 -19450.973} C_VEL
LIN {X 0,Y 270.592,Z 652.317,A -85,B 0,C 180,E1 -19451.908,E2 -19451.908} C_VEL
LIN {X 0,Y 273.175,Z 623.823,A -85,B 0,C 180,E1 -19453.118,E2 -19453.118} C_VEL
LIN {X 0,Y 269.754,Z 617.274,A -85,B 0,C 180,E1 -19454.682,E2 -19454.682} C_VEL
LIN {X 0,Y 265.449,Z 609.996,A -85,B 0,C 180,E1 -19456.885,E2 -19456.885} C_VEL
LIN {X 0,Y 263.21,Z 606.44,A -85,B 0,C 180,E1 -19458.185,E2 -19458.185} C_VEL
LIN {X 0,Y 261.506,Z 603.768,A -85,B 0,C 180,E1 -19459.267,E2 -19459.267} C_VEL
LIN {X 0,Y 259.065,Z 600.14,A -85,B 0,C 180,E1 -19461,E2 -19461} C_VEL
LIN {X 0,Y 257.726,Z 598.663,A -85,B 0,C 180,E1 -19462.01,E2 -19462.01} C_VEL
LIN {X 0,Y 256.477,Z 597.222,A -85,B 0,C 180,E1 -19463.074,E2 -19463.074} C_VEL
LIN {X 0,Y 253.712,Z 595.068,A -85,B 0,C 180,E1 -19465.845,E2 -19465.845} C_VEL
LIN {X 0,Y 251.897,Z 594.554,A -85,B 0,C 180,E1 -19468.314,E2 -19468.314} C_VEL
LIN {X 0,Y 250.738,Z 594.565,A -85,B 0,C 180,E1 -19471.326,E2 -19471.326} C_VEL
LIN {X 0,Y 250.529,Z 595.334,A -85,B 0,C 180,E1 -19473.776,E2 -19473.776} C_VEL
LIN {X 0,Y 251.077,Z 597.747,A -85,B 0,C 180,E1 -19476.701,E2 -19476.701} C_VEL
LIN {X 0,Y 252.055,Z 600.21,A -85,B 0,C 180,E1 -19478.832,E2 -19478.832} C_VEL
LIN {X 0,Y 254.671,Z 606.524,A -85,B 0,C 180,E1 -19482.36,E2 -19482.36} C_VEL
LIN {X 0,Y 257.306,Z 611.696,A -85,B 0,C 180,E1 -19484.755,E2 -19484.755} C_VEL
LIN {X 0,Y 261.03,Z 620.117,A -85,B 0,C 180,E1 -19487.516,E2 -19487.516} C_VEL
LIN {X 0,Y 264.048,Z 627.56,A -85,B 0,C 180,E1 -19489.442,E2 -19489.442} C_VEL
LIN {X 0,Y 266.319,Z 633.654,A -85,B 0,C 180,E1 -19490.747,E2 -19490.747} C_VEL
LIN {X 0,Y 266.766,Z 637.076,A -85,B 0,C 180,E1 -19491.163,E2 -19491.163} C_VEL
LIN {X 0,Y 267.831,Z 653.739,A -85,B 0,C 180,E1 -19492.731,E2 -19492.731} C_VEL
LIN {X 0,Y 268.305,Z 670.608,A -85,B 0,C 180,E1 -19494.004,E2 -19494.004} C_VEL
LIN {X 0,Y 268.16,Z 685.535,A -85,B 0,C 180,E1 -19494.938,E2 -19494.938} C_VEL
LIN {X 0,Y 267.658,Z 693.016,A -85,B 0,C 180,E1 -19495.283,E2 -19495.283} C_VEL
LIN {X 0,Y 265.411,Z 714.526,A -85,B 0,C 180,E1 -19496.144,E2 -19496.144} C_VEL
LIN {X 0,Y 263.096,Z 727.968,A -85,B 0,C 180,E1 -19496.913,E2 -19496.913} C_VEL
LIN {X 0,Y 259.948,Z 741.475,A -85,B 0,C 180,E1 -19497.957,E2 -19497.957} C_VEL
LIN {X 0,Y 256.298,Z 754.341,A -85,B 0,C 180,E1 -19499.29,E2 -19499.29} C_VEL
LIN {X 0,Y 252.055,Z 767.175,A -85,B 0,C 180,E1 -19501.025,E2 -19501.025} C_VEL
LIN {X 0,Y 248.933,Z 775.95,A -85,B 0,C 180,E1 -19502.466,E2 -19502.466} C_VEL
LIN {X 0,Y 247.119,Z 787.511,A -85,B 0,C 180,E1 -19503.619,E2 -19503.619} C_VEL
LIN {X 0,Y 245.139,Z 798.058,A -85,B 0,C 180,E1 -19504.986,E2 -19504.986} C_VEL
LIN {X 0,Y 242.768,Z 808.814,A -85,B 0,C 180,E1 -19506.771,E2 -19506.771} C_VEL
LIN {X 0,Y 240.706,Z 817.591,A -85,B 0,C 180,E1 -19508.596,E2 -19508.596} C_VEL
LIN {X 0,Y 238.802,Z 825.73,A -85,B 0,C 180,E1 -19510.688,E2 -19510.688} C_VEL
LIN {X 0,Y 236.835,Z 833.56,A -85,B 0,C 180,E1 -19513.184,E2 -19513.184} C_VEL
LIN {X 0,Y 235.394,Z 838.891,A -85,B 0,C 180,E1 -19515.3,E2 -19515.3} C_VEL
LIN {X 0,Y 234.218,Z 844.102,A -85,B 0,C 180,E1 -19517.877,E2 -19517.877} C_VEL
LIN {X 0,Y 233.415,Z 848.133,A -85,B 0,C 180,E1 -19520.469,E2 -19520.469} C_VEL
LIN {X 0,Y 232.922,Z 851.103,A -85,B 0,C 180,E1 -19523.069,E2 -19523.069} C_VEL
LIN {X 0,Y 232.794,Z 852.687,A -85,B 0,C 180,E1 -19525.047,E2 -19525.047} C_VEL
LIN {X 0,Y 232.84,Z 854.154,A -85,B 0,C 180,E1 -19528.272,E2 -19528.272} C_VEL
LIN {X 0,Y 232.925,Z 854.373,A -85,B 0,C 180,E1 -19530.001,E2 -19530.001} C_VEL
LIN {X 0,Y 232.83,Z 854.143,A -85,B 0,C 180,E1 -19531.731,E2 -19531.731} C_VEL
LIN {X 0,Y 232.842,Z 852.503,A -85,B 0,C 180,E1 -19535.197,E2 -19535.197} C_VEL
LIN {X 0,Y 232.927,Z 851.061,A -85,B 0,C 180,E1 -19536.933,E2 -19536.933} C_VEL
LIN {X 0,Y 233.426,Z 848.076,A -85,B 0,C 180,E1 -19539.533,E2 -19539.533} C_VEL
LIN {X 0,Y 234.174,Z 844.027,A -85,B 0,C 180,E1 -19542.128,E2 -19542.128} C_VEL
LIN {X 0,Y 235.645,Z 837.787,A -85,B 0,C 180,E1 -19545.129,E2 -19545.129} C_VEL
LIN {X 0,Y 237.361,Z 830.985,A -85,B 0,C 180,E1 -19547.669,E2 -19547.669} C_VEL
LIN {X 0,Y 239.408,Z 822.937,A -85,B 0,C 180,E1 -19550.051,E2 -19550.051} C_VEL
LIN {X 0,Y 241.52,Z 813.716,A -85,B 0,C 180,E1 -19552.229,E2 -19552.229} C_VEL
LIN {X 0,Y 243.791,Z 804.097,A -85,B 0,C 180,E1 -19554.03,E2 -19554.03} C_VEL
LIN {X 0,Y 245.979,Z 793.557,A -85,B 0,C 180,E1 -19555.605,E2 -19555.605} C_VEL
LIN {X 0,Y 247.952,Z 781.743,A -85,B 0,C 180,E1 -19556.97,E2 -19556.97} C_VEL
LIN {X 0,Y 249.705,Z 769.484,A -85,B 0,C 180,E1 -19558.014,E2 -19558.014} C_VEL
LIN {X 0,Y 251.133,Z 757.008,A -85,B 0,C 180,E1 -19558.74,E2 -19558.74} C_VEL
LIN {X 0,Y 251.932,Z 742.732,A -85,B 0,C 180,E1 -19559.247,E2 -19559.247} C_VEL
LIN {X 0,Y 253.789,Z 687.04,A -85,B 0,C 180,E1 -19560.786,E2 -19560.786} C_VEL
LIN {X 0,Y 251.254,Z 659.328,A -85,B 0,C 180,E1 -19562.036,E2 -19562.036} C_VEL
LIN {X 0,Y 247.965,Z 634.26,A -85,B 0,C 180,E1 -19563.359,E2 -19563.359} C_VEL
LIN {X 0,Y 247.849,Z 611.544,A -85,B 0,C 180,E1 -19566.086,E2 -19566.086} C_VEL
LIN {X 0,Y 244.041,Z 598.705,A -85,B 0,C 180,E1 -19568.292,E2 -19568.292} C_VEL
LIN {X 0,Y 240.011,Z 585.652,A -85,B 0,C 180,E1 -19570.797,E2 -19570.797} C_VEL
LIN {X 0,Y 236.872,Z 576.226,A -85,B 0,C 180,E1 -19572.766,E2 -19572.766} C_VEL
LIN {X 0,Y 234.978,Z 571.735,A -85,B 0,C 180,E1 -19573.884,E2 -19573.884} C_VEL
LIN {X 0,Y 234.9,Z 571.211,A -85,B 0,C 180,E1 -19574.03,E2 -19574.03} C_VEL
LIN {X 0,Y 234.887,Z 571.21,A -85,B 0,C 180,E1 -19578.42,E2 -19578.42} C_VEL
LIN {X 0,Y 234.921,Z 571.222,A -85,B 0,C 180,E1 -19581.079,E2 -19581.079} C_VEL
LIN {X 0,Y 234.929,Z 571.217,A -85,B 0,C 180,E1 -19585.362,E2 -19585.362} C_VEL
LIN {X 0,Y 234.934,Z 571.198,A -85,B 0,C 180,E1 -19589.433,E2 -19589.433} C_VEL
LIN {X 0,Y 234.997,Z 571.196,A -85,B 0,C 180,E1 -19593.794,E2 -19593.794} C_VEL
LIN {X 0,Y 235.001,Z 571.214,A -85,B 0,C 180,E1 -19598.969,E2 -19598.969} C_VEL
LIN {X 0,Y 235.099,Z 571.172,A -85,B 0,C 180,E1 -19603.06,E2 -19603.06} C_VEL
LIN {X 0,Y 235.116,Z 571.178,A -85,B 0,C 180,E1 -19607.922,E2 -19607.922} C_VEL
LIN {X 0,Y 235.334,Z 571.152,A -85,B 0,C 180,E1 -19611.413,E2 -19611.413} C_VEL
LIN {X 0,Y 235.376,Z 571.165,A -85,B 0,C 180,E1 -19613.141,E2 -19613.141} C_VEL
LIN {X 0,Y 235.597,Z 571.108,A -85,B 0,C 180,E1 -19618.291,E2 -19618.291} C_VEL
LIN {X 0,Y 235.598,Z 571.137,A -85,B 0,C 180,E1 -19621.71,E2 -19621.71} C_VEL
LIN {X 0,Y 235.405,Z 571.143,A -85,B 0,C 180,E1 -19626.859,E2 -19626.859} C_VEL
LIN {X 0,Y 235.241,Z 571.171,A -85,B 0,C 180,E1 -19630.326,E2 -19630.326} C_VEL
LIN {X 0,Y 235.115,Z 571.198,A -85,B 0,C 180,E1 -19635.606,E2 -19635.606} C_VEL
LIN {X 0,Y 235.011,Z 571.184,A -85,B 0,C 180,E1 -19639.206,E2 -19639.206} C_VEL
LIN {X 0,Y 234.964,Z 571.216,A -85,B 0,C 180,E1 -19642.883,E2 -19642.883} C_VEL
LIN {X 0,Y 234.973,Z 571.201,A -85,B 0,C 180,E1 -19646.657,E2 -19646.657} C_VEL
LIN {X 0,Y 234.934,Z 571.203,A -85,B 0,C 180,E1 -19650.568,E2 -19650.568} C_VEL
LIN {X 0,Y 234.937,Z 571.212,A -85,B 0,C 180,E1 -19654.637,E2 -19654.637} C_VEL
LIN {X 0,Y 234.945,Z 571.213,A -85,B 0,C 180,E1 -19658.944,E2 -19658.944} C_VEL
LIN {X 0,Y 234.945,Z 571.335,A -85,B 0,C 180,E1 -19660.236,E2 -19660.236} C_VEL
LIN {X 0,Y 238.241,Z 579.582,A -85,B 0,C 180,E1 -19663.304,E2 -19663.304} C_VEL
LIN {X 0,Y 242.22,Z 590.56,A -85,B 0,C 180,E1 -19667.07,E2 -19667.07} C_VEL
LIN {X 0,Y 245.673,Z 601.913,A -85,B 0,C 180,E1 -19670.57,E2 -19670.57} C_VEL
LIN {X 0,Y 248.486,Z 613.525,A -85,B 0,C 180,E1 -19673.821,E2 -19673.821} C_VEL
LIN {X 0,Y 250.081,Z 621.229,A -85,B 0,C 180,E1 -19675.801,E2 -19675.801} C_VEL
LIN {X 0,Y 249.731,Z 625.742,A -85,B 0,C 180,E1 -19676.715,E2 -19676.715} C_VEL
LIN {X 0,Y 249.949,Z 628.042,A -85,B 0,C 180,E1 -19676.917,E2 -19676.917} C_VEL
LIN {X 0,Y 254.148,Z 655.491,A -85,B 0,C 180,E1 -19678.434,E2 -19678.434} C_VEL
LIN {X 0,Y 255.163,Z 663.019,A -85,B 0,C 180,E1 -19678.819,E2 -19678.819} C_VEL
LIN {X 0,Y 252.322,Z 738.923,A -85,B 0,C 180,E1 -19680.941,E2 -19680.941} C_VEL
LIN {X 0,Y 251.273,Z 752.138,A -85,B 0,C 180,E1 -19681.608,E2 -19681.608} C_VEL
LIN {X 0,Y 249.765,Z 764.645,A -85,B 0,C 180,E1 -19682.562,E2 -19682.562} C_VEL
LIN {X 0,Y 248.058,Z 775.868,A -85,B 0,C 180,E1 -19683.723,E2 -19683.723} C_VEL
LIN {X 0,Y 245.807,Z 787.469,A -85,B 0,C 180,E1 -19685.281,E2 -19685.281} C_VEL
LIN {X 0,Y 243.549,Z 798.229,A -85,B 0,C 180,E1 -19687.161,E2 -19687.161} C_VEL
LIN {X 0,Y 241.502,Z 807.474,A -85,B 0,C 180,E1 -19689.198,E2 -19689.198} C_VEL
LIN {X 0,Y 239.203,Z 816.138,A -85,B 0,C 180,E1 -19691.587,E2 -19691.587} C_VEL
LIN {X 0,Y 237.223,Z 823.354,A -85,B 0,C 180,E1 -19694.094,E2 -19694.094} C_VEL
LIN {X 0,Y 235.404,Z 829.973,A -85,B 0,C 180,E1 -19697.06,E2 -19697.06} C_VEL
LIN {X 0,Y 234.316,Z 834.311,A -85,B 0,C 180,E1 -19699.631,E2 -19699.631} C_VEL
LIN {X 0,Y 233.793,Z 836.592,A -85,B 0,C 180,E1 -19701.354,E2 -19701.354} C_VEL
LIN {X 0,Y 233.226,Z 839.197,A -85,B 0,C 180,E1 -19703.945,E2 -19703.945} C_VEL
LIN {X 0,Y 232.918,Z 840.862,A -85,B 0,C 180,E1 -19706.539,E2 -19706.539} C_VEL
LIN {X 0,Y 232.833,Z 841.705,A -85,B 0,C 180,E1 -19709.999,E2 -19709.999} C_VEL
LIN {X 0,Y 232.828,Z 841.51,A -85,B 0,C 180,E1 -19711.728,E2 -19711.728} C_VEL
LIN {X 0,Y 232.915,Z 840.922,A -85,B 0,C 180,E1 -19713.458,E2 -19713.458} C_VEL
LIN {X 0,Y 233.235,Z 839.286,A -85,B 0,C 180,E1 -19716.075,E2 -19716.075} C_VEL
LIN {X 0,Y 234.007,Z 835.703,A -85,B 0,C 180,E1 -19719.506,E2 -19719.506} C_VEL
LIN {X 0,Y 234.972,Z 831.785,A -85,B 0,C 180,E1 -19722.084,E2 -19722.084} C_VEL
LIN {X 0,Y 236.34,Z 826.71,A -85,B 0,C 180,E1 -19724.639,E2 -19724.639} C_VEL
LIN {X 0,Y 238.041,Z 820.311,A -85,B 0,C 180,E1 -19727.17,E2 -19727.17} C_VEL
LIN {X 0,Y 240.29,Z 812.34,A -85,B 0,C 180,E1 -19729.653,E2 -19729.653} C_VEL
LIN {X 0,Y 242.441,Z 803.585,A -85,B 0,C 180,E1 -19731.84,E2 -19731.84} C_VEL
LIN {X 0,Y 244.508,Z 794.156,A -85,B 0,C 180,E1 -19733.727,E2 -19733.727} C_VEL
LIN {X 0,Y 246.582,Z 784.251,A -85,B 0,C 180,E1 -19735.309,E2 -19735.309} C_VEL
LIN {X 0,Y 248.555,Z 773.474,A -85,B 0,C 180,E1 -19736.669,E2 -19736.669} C_VEL
LIN {X 0,Y 250.269,Z 761.577,A -85,B 0,C 180,E1 -19737.829,E2 -19737.829} C_VEL
LIN {X 0,Y 251.603,Z 749.226,A -85,B 0,C 180,E1 -19738.69,E2 -19738.69} C_VEL
LIN {X 0,Y 252.578,Z 735.426,A -85,B 0,C 180,E1 -19739.309,E2 -19739.309} C_VEL
LIN {X 0,Y 255.149,Z 665.868,A -85,B 0,C 180,E1 -19741.224,E2 -19741.224} C_VEL
LIN {X 0,Y 250.704,Z 638.513,A -85,B 0,C 180,E1 -19742.754,E2 -19742.754} C_VEL
LIN {X 0,Y 248.528,Z 626.842,A -85,B 0,C 180,E1 -19743.506,E2 -19743.506} C_VEL
LIN {X 0,Y 249.181,Z 621.078,A -85,B 0,C 180,E1 -19744.801,E2 -19744.801} C_VEL
LIN {X 0,Y 247.151,Z 610.278,A -85,B 0,C 180,E1 -19747.899,E2 -19747.899} C_VEL
LIN {X 0,Y 244.484,Z 599.244,A -85,B 0,C 180,E1 -19751.386,E2 -19751.386} C_VEL
LIN {X 0,Y 244.062,Z 597.588,A -85,B 0,C 180,E1 -19751.976,E2 -19751.976} C_VEL
LIN {X 0,Y 245.247,Z 599.756,A -85,B 0,C 180,E1 -19752.147,E2 -19752.147} C_VEL
LIN {X 0,Y 243.818,Z 645.445,A -85,B 0,C 180,E1 -19753.923,E2 -19753.923} C_VEL
LIN {X 0,Y 243.504,Z 659.971,A -85,B 0,C 180,E1 -19754.632,E2 -19754.632} C_VEL
LIN {X 0,Y 242.769,Z 674.416,A -85,B 0,C 180,E1 -19755.701,E2 -19755.701} C_VEL
LIN {X 0,Y 241.817,Z 687.871,A -85,B 0,C 180,E1 -19757.089,E2 -19757.089} C_VEL
LIN {X 0,Y 240.797,Z 699.598,A -85,B 0,C 180,E1 -19758.643,E2 -19758.643} C_VEL
LIN {X 0,Y 239.576,Z 711.418,A -85,B 0,C 180,E1 -19760.626,E2 -19760.626} C_VEL
LIN {X 0,Y 238.449,Z 721.508,A -85,B 0,C 180,E1 -19762.727,E2 -19762.727} C_VEL
LIN {X 0,Y 237.512,Z 729.545,A -85,B 0,C 180,E1 -19764.759,E2 -19764.759} C_VEL
LIN {X 0,Y 236.595,Z 737.42,A -85,B 0,C 180,E1 -19767.183,E2 -19767.183} C_VEL
LIN {X 0,Y 236.016,Z 744.087,A -85,B 0,C 180,E1 -19769.713,E2 -19769.713} C_VEL
LIN {X 0,Y 235.549,Z 749.864,A -85,B 0,C 180,E1 -19772.453,E2 -19772.453} C_VEL
LIN {X 0,Y 235.35,Z 754.444,A -85,B 0,C 180,E1 -19775.287,E2 -19775.287} C_VEL
LIN {X 0,Y 235.496,Z 757.297,A -85,B 0,C 180,E1 -19777.684,E2 -19777.684} C_VEL
LIN {X 0,Y 236.16,Z 759.771,A -85,B 0,C 180,E1 -19780.892,E2 -19780.892} C_VEL
LIN {X 0,Y 236.352,Z 760.115,A -85,B 0,C 180,E1 -19781.604,E2 -19781.604} C_VEL
LIN {X 0,Y 236.167,Z 760.744,A -85,B 0,C 180,E1 -19783.028,E2 -19783.028} C_VEL
LIN {X 0,Y 234.331,Z 761.413,A -85,B 0,C 180,E1 -19785.395,E2 -19785.395} C_VEL
LIN {X 0,Y 232.798,Z 761.456,A -85,B 0,C 180,E1 -19787.8,E2 -19787.8} C_VEL
LIN {X 0,Y 233.089,Z 760.898,A -85,B 0,C 180,E1 -19789.248,E2 -19789.248} C_VEL
LIN {X 0,Y 234.669,Z 759.437,A -85,B 0,C 180,E1 -19791.388,E2 -19791.388} C_VEL
LIN {X 0,Y 237.034,Z 756.557,A -85,B 0,C 180,E1 -19794.043,E2 -19794.043} C_VEL
LIN {X 0,Y 239.798,Z 752.498,A -85,B 0,C 180,E1 -19796.64,E2 -19796.64} C_VEL
LIN {X 0,Y 243.421,Z 746.153,A -85,B 0,C 180,E1 -19799.586,E2 -19799.586} C_VEL
LIN {X 0,Y 246.875,Z 739.298,A -85,B 0,C 180,E1 -19801.991,E2 -19801.991} C_VEL
LIN {X 0,Y 250.066,Z 731.95,A -85,B 0,C 180,E1 -19804.029,E2 -19804.029} C_VEL
LIN {X 0,Y 253.313,Z 723.236,A -85,B 0,C 180,E1 -19805.972,E2 -19805.972} C_VEL
LIN {X 0,Y 256.796,Z 712.612,A -85,B 0,C 180,E1 -19807.865,E2 -19807.865} C_VEL
LIN {X 0,Y 259.631,Z 702.037,A -85,B 0,C 180,E1 -19809.347,E2 -19809.347} C_VEL
LIN {X 0,Y 262.092,Z 690.508,A -85,B 0,C 180,E1 -19810.623,E2 -19810.623} C_VEL
LIN {X 0,Y 264.138,Z 677.343,A -85,B 0,C 180,E1 -19811.754,E2 -19811.754} C_VEL
LIN {X 0,Y 265.536,Z 663.94,A -85,B 0,C 180,E1 -19812.583,E2 -19812.583} C_VEL
LIN {X 0,Y 267.689,Z 638.793,A -85,B 0,C 180,E1 -19813.743,E2 -19813.743} C_VEL
LIN {X 0,Y 268.869,Z 627.135,A -85,B 0,C 180,E1 -19814.235,E2 -19814.235} C_VEL
LIN {X 0,Y 264.937,Z 619.773,A -85,B 0,C 180,E1 -19816.235,E2 -19816.235} C_VEL
LIN {X 0,Y 261.034,Z 613.043,A -85,B 0,C 180,E1 -19818.533,E2 -19818.533} C_VEL
LIN {X 0,Y 259.063,Z 610.043,A -85,B 0,C 180,E1 -19819.803,E2 -19819.803} C_VEL
LIN {X 0,Y 256.364,Z 605.882,A -85,B 0,C 180,E1 -19821.906,E2 -19821.906} C_VEL
LIN {X 0,Y 254.838,Z 604.108,A -85,B 0,C 180,E1 -19823.232,E2 -19823.232} C_VEL
LIN {X 0,Y 252.173,Z 601.983,A -85,B 0,C 180,E1 -19826.015,E2 -19826.015} C_VEL
LIN {X 0,Y 250.014,Z 601.414,A -85,B 0,C 180,E1 -19829.38,E2 -19829.38} C_VEL
LIN {X 0,Y 249.145,Z 602.022,A -85,B 0,C 180,E1 -19833.26,E2 -19833.26} C_VEL
LIN {X 0,Y 249.69,Z 604.889,A -85,B 0,C 180,E1 -19836.749,E2 -19836.749} C_VEL
LIN {X 0,Y 250.522,Z 607.232,A -85,B 0,C 180,E1 -19838.671,E2 -19838.671} C_VEL
LIN {X 0,Y 253.315,Z 614.319,A -85,B 0,C 180,E1 -19842.522,E2 -19842.522} C_VEL
LIN {X 0,Y 254.999,Z 617.882,A -85,B 0,C 180,E1 -19844.141,E2 -19844.141} C_VEL
LIN {X 0,Y 258.233,Z 625.75,A -85,B 0,C 180,E1 -19846.784,E2 -19846.784} C_VEL
LIN {X 0,Y 260.961,Z 632.886,A -85,B 0,C 180,E1 -19848.664,E2 -19848.664} C_VEL
LIN {X 0,Y 262.747,Z 638.198,A -85,B 0,C 180,E1 -19849.848,E2 -19849.848} C_VEL
LIN {X 0,Y 263.64,Z 654.123,A -85,B 0,C 180,E1 -19851.412,E2 -19851.412} C_VEL
LIN {X 0,Y 263.966,Z 670.735,A -85,B 0,C 180,E1 -19852.759,E2 -19852.759} C_VEL
LIN {X 0,Y 263.687,Z 686.972,A -85,B 0,C 180,E1 -19853.787,E2 -19853.787} C_VEL
LIN {X 0,Y 263.235,Z 693.255,A -85,B 0,C 180,E1 -19854.082,E2 -19854.082} C_VEL
LIN {X 0,Y 260.887,Z 713.698,A -85,B 0,C 180,E1 -19854.929,E2 -19854.929} C_VEL
LIN {X 0,Y 258.286,Z 727.526,A -85,B 0,C 180,E1 -19855.745,E2 -19855.745} C_VEL
LIN {X 0,Y 255.027,Z 740.767,A -85,B 0,C 180,E1 -19856.792,E2 -19856.792} C_VEL
LIN {X 0,Y 251.212,Z 753.501,A -85,B 0,C 180,E1 -19858.128,E2 -19858.128} C_VEL
LIN {X 0,Y 247.218,Z 765.059,A -85,B 0,C 180,E1 -19859.697,E2 -19859.697} C_VEL
LIN {X 0,Y 243.059,Z 775.618,A -85,B 0,C 180,E1 -19861.506,E2 -19861.506} C_VEL
LIN {X 0,Y 242.414,Z 777.447,A -85,B 0,C 180,E1 -19861.836,E2 -19861.836} C_VEL
LIN {X 0,Y 240.456,Z 789.018,A -85,B 0,C 180,E1 -19863.064,E2 -19863.064} C_VEL
LIN {X 0,Y 238.129,Z 800.454,A -85,B 0,C 180,E1 -19864.665,E2 -19864.665} C_VEL
LIN {X 0,Y 235.756,Z 810.75,A -85,B 0,C 180,E1 -19866.504,E2 -19866.504} C_VEL
LIN {X 0,Y 233.679,Z 819.177,A -85,B 0,C 180,E1 -19868.383,E2 -19868.383} C_VEL
LIN {X 0,Y 231.748,Z 826.939,A -85,B 0,C 180,E1 -19870.515,E2 -19870.515} C_VEL
LIN {X 0,Y 229.71,Z 834.495,A -85,B 0,C 180,E1 -19873.105,E2 -19873.105} C_VEL
LIN {X 0,Y 227.973,Z 840.557,A -85,B 0,C 180,E1 -19875.724,E2 -19875.724} C_VEL
LIN {X 0,Y 226.906,Z 845.354,A -85,B 0,C 180,E1 -19878.387,E2 -19878.387} C_VEL
LIN {X 0,Y 226.17,Z 849.021,A -85,B 0,C 180,E1 -19881.063,E2 -19881.063} C_VEL
LIN {X 0,Y 225.847,Z 850.91,A -85,B 0,C 180,E1 -19882.851,E2 -19882.851} C_VEL
LIN {X 0,Y 225.714,Z 852.641,A -85,B 0,C 180,E1 -19885.123,E2 -19885.123} C_VEL
LIN {X 0,Y 225.75,Z 853.961,A -85,B 0,C 180,E1 -19888.218,E2 -19888.218} C_VEL
LIN {X 0,Y 225.832,Z 854.18,A -85,B 0,C 180,E1 -19890.001,E2 -19890.001} C_VEL
LIN {X 0,Y 225.741,Z 853.95,A -85,B 0,C 180,E1 -19891.786,E2 -19891.786} C_VEL
LIN {X 0,Y 225.745,Z 852.309,A -85,B 0,C 180,E1 -19895.36,E2 -19895.36} C_VEL
LIN {X 0,Y 225.853,Z 850.867,A -85,B 0,C 180,E1 -19897.152,E2 -19897.152} C_VEL
LIN {X 0,Y 226.38,Z 847.882,A -85,B 0,C 180,E1 -19899.833,E2 -19899.833} C_VEL
LIN {X 0,Y 227.204,Z 843.833,A -85,B 0,C 180,E1 -19902.507,E2 -19902.507} C_VEL
LIN {X 0,Y 228.763,Z 837.594,A -85,B 0,C 180,E1 -19905.595,E2 -19905.595} C_VEL
LIN {X 0,Y 230.58,Z 830.793,A -85,B 0,C 180,E1 -19908.206,E2 -19908.206} C_VEL
LIN {X 0,Y 232.58,Z 823.358,A -85,B 0,C 180,E1 -19910.488,E2 -19910.488} C_VEL
LIN {X 0,Y 234.479,Z 815.457,A -85,B 0,C 180,E1 -19912.468,E2 -19912.468} C_VEL
LIN {X 0,Y 237.047,Z 805.073,A -85,B 0,C 180,E1 -19914.525,E2 -19914.525} C_VEL
LIN {X 0,Y 239.293,Z 794.792,A -85,B 0,C 180,E1 -19916.14,E2 -19916.14} C_VEL
LIN {X 0,Y 241.366,Z 783.504,A -85,B 0,C 180,E1 -19917.533,E2 -19917.533} C_VEL
LIN {X 0,Y 243.312,Z 770.585,A -85,B 0,C 180,E1 -19918.7,E2 -19918.7} C_VEL
LIN {X 0,Y 244.745,Z 758.705,A -85,B 0,C 180,E1 -19919.445,E2 -19919.445} C_VEL
LIN {X 0,Y 245.634,Z 746.46,A -85,B 0,C 180,E1 -19919.942,E2 -19919.942} C_VEL
LIN {X 0,Y 247.717,Z 688.106,A -85,B 0,C 180,E1 -19921.588,E2 -19921.588} C_VEL
LIN {X 0,Y 245.29,Z 660.606,A -85,B 0,C 180,E1 -19922.866,E2 -19922.866} C_VEL
LIN {X 0,Y 241.896,Z 634.176,A -85,B 0,C 180,E1 -19924.308,E2 -19924.308} C_VEL
LIN {X 0,Y 242.039,Z 615.329,A -85,B 0,C 180,E1 -19926.646,E2 -19926.646} C_VEL
LIN {X 0,Y 241.413,Z 612.173,A -85,B 0,C 180,E1 -19927.161,E2 -19927.161} C_VEL
LIN {X 0,Y 237.429,Z 598.347,A -85,B 0,C 180,E1 -19929.681,E2 -19929.681} C_VEL
LIN {X 0,Y 234.653,Z 589.296,A -85,B 0,C 180,E1 -19931.516,E2 -19931.516} C_VEL
LIN {X 0,Y 231.925,Z 580.746,A -85,B 0,C 180,E1 -19933.342,E2 -19933.342} C_VEL
LIN {X 0,Y 230.475,Z 577.391,A -85,B 0,C 180,E1 -19934.227,E2 -19934.227} C_VEL
LIN {X 0,Y 228.236,Z 573.689,A -85,B 0,C 180,E1 -19935.436,E2 -19935.436} C_VEL
LIN {X 0,Y 227.863,Z 572.1,A -85,B 0,C 180,E1 -19935.822,E2 -19935.822} C_VEL
LIN {X 0,Y 227.855,Z 572.103,A -85,B 0,C 180,E1 -19940.454,E2 -19940.454} C_VEL
LIN {X 0,Y 227.882,Z 572.081,A -85,B 0,C 180,E1 -19944.128,E2 -19944.128} C_VEL
LIN {X 0,Y 227.873,Z 572.078,A -85,B 0,C 180,E1 -19948.378,E2 -19948.378} C_VEL
LIN {X 0,Y 227.889,Z 572.098,A -85,B 0,C 180,E1 -19952.445,E2 -19952.445} C_VEL
LIN {X 0,Y 227.909,Z 572.073,A -85,B 0,C 180,E1 -19956.367,E2 -19956.367} C_VEL
LIN {X 0,Y 227.94,Z 572.078,A -85,B 0,C 180,E1 -19960.174,E2 -19960.174} C_VEL
LIN {X 0,Y 228.057,Z 572.058,A -85,B 0,C 180,E1 -19963.898,E2 -19963.898} C_VEL
LIN {X 0,Y 228.074,Z 572.06,A -85,B 0,C 180,E1 -19967.543,E2 -19967.543} C_VEL
LIN {X 0,Y 228.27,Z 572.027,A -85,B 0,C 180,E1 -19971.145,E2 -19971.145} C_VEL
LIN {X 0,Y 228.327,Z 572.042,A -85,B 0,C 180,E1 -19972.928,E2 -19972.928} C_VEL
LIN {X 0,Y 228.556,Z 571.984,A -85,B 0,C 180,E1 -19978.238,E2 -19978.238} C_VEL
LIN {X 0,Y 228.556,Z 572.014,A -85,B 0,C 180,E1 -19981.762,E2 -19981.762} C_VEL
LIN {X 0,Y 228.356,Z 572.024,A -85,B 0,C 180,E1 -19987.072,E2 -19987.072} C_VEL
LIN {X 0,Y 228.162,Z 572.047,A -85,B 0,C 180,E1 -19990.651,E2 -19990.651} C_VEL
LIN {X 0,Y 228.065,Z 572.06,A -85,B 0,C 180,E1 -19994.272,E2 -19994.272} C_VEL
LIN {X 0,Y 228.006,Z 572.064,A -85,B 0,C 180,E1 -19997.953,E2 -19997.953} C_VEL
LIN {X 0,Y 227.934,Z 572.094,A -85,B 0,C 180,E1 -20002.329,E2 -20002.329} C_VEL
LIN {X 0,Y 227.946,Z 572.075,A -85,B 0,C 180,E1 -20006.603,E2 -20006.603} C_VEL
LIN {X 0,Y 227.912,Z 572.078,A -85,B 0,C 180,E1 -20010.296,E2 -20010.296} C_VEL
LIN {X 0,Y 227.881,Z 572.1,A -85,B 0,C 180,E1 -20013.72,E2 -20013.72} C_VEL
LIN {X 0,Y 227.881,Z 572.097,A -85,B 0,C 180,E1 -20018.455,E2 -20018.455} C_VEL
LIN {X 0,Y 228.511,Z 574.238,A -85,B 0,C 180,E1 -20019.283,E2 -20019.283} C_VEL
LIN {X 0,Y 230.834,Z 579.512,A -85,B 0,C 180,E1 -20021.468,E2 -20021.468} C_VEL
LIN {X 0,Y 234.325,Z 588.637,A -85,B 0,C 180,E1 -20024.816,E2 -20024.816} C_VEL
LIN {X 0,Y 237.293,Z 597.334,A -85,B 0,C 180,E1 -20027.769,E2 -20027.769} C_VEL
LIN {X 0,Y 240.446,Z 608.549,A -85,B 0,C 180,E1 -20031.195,E2 -20031.195} C_VEL
LIN {X 0,Y 243.064,Z 620.196,A -85,B 0,C 180,E1 -20034.416,E2 -20034.416} C_VEL
LIN {X 0,Y 243.783,Z 624.724,A -85,B 0,C 180,E1 -20035.533,E2 -20035.533} C_VEL
LIN {X 0,Y 243.567,Z 626.487,A -85,B 0,C 180,E1 -20035.876,E2 -20035.876} C_VEL
LIN {X 0,Y 248.092,Z 656.256,A -85,B 0,C 180,E1 -20037.594,E2 -20037.594} C_VEL
LIN {X 0,Y 249.084,Z 664.763,A -85,B 0,C 180,E1 -20038.024,E2 -20038.024} C_VEL
LIN {X 0,Y 246.153,Z 739.056,A -85,B 0,C 180,E1 -20040.14,E2 -20040.14} C_VEL
LIN {X 0,Y 245.065,Z 752.302,A -85,B 0,C 180,E1 -20040.821,E2 -20040.821} C_VEL
LIN {X 0,Y 243.491,Z 764.82,A -85,B 0,C 180,E1 -20041.793,E2 -20041.793} C_VEL
LIN {X 0,Y 241.717,Z 776.049,A -85,B 0,C 180,E1 -20042.979,E2 -20042.979} C_VEL
LIN {X 0,Y 239.386,Z 787.654,A -85,B 0,C 180,E1 -20044.571,E2 -20044.571} C_VEL
LIN {X 0,Y 236.877,Z 799.042,A -85,B 0,C 180,E1 -20046.619,E2 -20046.619} C_VEL
LIN {X 0,Y 234.838,Z 807.788,A -85,B 0,C 180,E1 -20048.613,E2 -20048.613} C_VEL
LIN {X 0,Y 232.462,Z 816.33,A -85,B 0,C 180,E1 -20051.033,E2 -20051.033} C_VEL
LIN {X 0,Y 230.373,Z 823.547,A -85,B 0,C 180,E1 -20053.608,E2 -20053.608} C_VEL
LIN {X 0,Y 228.484,Z 830.166,A -85,B 0,C 180,E1 -20056.661,E2 -20056.661} C_VEL
LIN {X 0,Y 227.318,Z 834.505,A -85,B 0,C 180,E1 -20059.308,E2 -20059.308} C_VEL
LIN {X 0,Y 226.768,Z 836.785,A -85,B 0,C 180,E1 -20061.084,E2 -20061.084} C_VEL
LIN {X 0,Y 226.109,Z 839.638,A -85,B 0,C 180,E1 -20064.066,E2 -20064.066} C_VEL
LIN {X 0,Y 225.828,Z 841.056,A -85,B 0,C 180,E1 -20066.43,E2 -20066.43} C_VEL
LIN {X 0,Y 225.747,Z 841.667,A -85,B 0,C 180,E1 -20068.215,E2 -20068.215} C_VEL
LIN {X 0,Y 225.746,Z 841.898,A -85,B 0,C 180,E1 -20069.999,E2 -20069.999} C_VEL
LIN {X 0,Y 225.745,Z 841.702,A -85,B 0,C 180,E1 -20071.783,E2 -20071.783} C_VEL
LIN {X 0,Y 226.011,Z 840.146,A -85,B 0,C 180,E1 -20075.351,E2 -20075.351} C_VEL
LIN {X 0,Y 226.322,Z 838.775,A -85,B 0,C 180,E1 -20077.134,E2 -20077.134} C_VEL
LIN {X 0,Y 227.002,Z 835.894,A -85,B 0,C 180,E1 -20079.802,E2 -20079.802} C_VEL
LIN {X 0,Y 228.025,Z 831.976,A -85,B 0,C 180,E1 -20082.458,E2 -20082.458} C_VEL
LIN {X 0,Y 229.476,Z 826.899,A -85,B 0,C 180,E1 -20085.088,E2 -20085.088} C_VEL
LIN {X 0,Y 231.277,Z 820.499,A -85,B 0,C 180,E1 -20087.689,E2 -20087.689} C_VEL
LIN {X 0,Y 233.627,Z 812.526,A -85,B 0,C 180,E1 -20090.238,E2 -20090.238} C_VEL
LIN {X 0,Y 235.944,Z 803.367,A -85,B 0,C 180,E1 -20092.572,E2 -20092.572} C_VEL
LIN {X 0,Y 238.282,Z 793.196,A -85,B 0,C 180,E1 -20094.619,E2 -20094.619} C_VEL
LIN {X 0,Y 240.506,Z 783.045,A -85,B 0,C 180,E1 -20096.228,E2 -20096.228} C_VEL
LIN {X 0,Y 242.506,Z 771.911,A -85,B 0,C 180,E1 -20097.624,E2 -20097.624} C_VEL
LIN {X 0,Y 244.193,Z 760.508,A -85,B 0,C 180,E1 -20098.701,E2 -20098.701} C_VEL
LIN {X 0,Y 245.487,Z 748.512,A -85,B 0,C 180,E1 -20099.533,E2 -20099.533} C_VEL
LIN {X 0,Y 246.432,Z 735.516,A -85,B 0,C 180,E1 -20100.114,E2 -20100.114} C_VEL
LIN {X 0,Y 249.027,Z 666.43,A -85,B 0,C 180,E1 -20102.064,E2 -20102.064} C_VEL
LIN {X 0,Y 244.515,Z 638.609,A -85,B 0,C 180,E1 -20103.691,E2 -20103.691} C_VEL
LIN {X 0,Y 242.395,Z 627.034,A -85,B 0,C 180,E1 -20104.468,E2 -20104.468} C_VEL
LIN {X 0,Y 242.755,Z 623.09,A -85,B 0,C 180,E1 -20105.379,E2 -20105.379} C_VEL
LIN {X 0,Y 240.825,Z 612.885,A -85,B 0,C 180,E1 -20108.377,E2 -20108.377} C_VEL
LIN {X 0,Y 238.33,Z 602.438,A -85,B 0,C 180,E1 -20111.735,E2 -20111.735} C_VEL
LIN {X 0,Y 236.927,Z 647.582,A -85,B 0,C 180,E1 -20113.591,E2 -20113.591} C_VEL
LIN {X 0,Y 236.55,Z 661.713,A -85,B 0,C 180,E1 -20114.328,E2 -20114.328} C_VEL
LIN {X 0,Y 235.806,Z 675.759,A -85,B 0,C 180,E1 -20115.417,E2 -20115.417} C_VEL
LIN {X 0,Y 234.834,Z 688.686,A -85,B 0,C 180,E1 -20116.796,E2 -20116.796} C_VEL
LIN {X 0,Y 233.835,Z 699.897,A -85,B 0,C 180,E1 -20118.319,E2 -20118.319} C_VEL
LIN {X 0,Y 232.716,Z 710.399,A -85,B 0,C 180,E1 -20120.077,E2 -20120.077} C_VEL
LIN {X 0,Y 231.573,Z 720.692,A -85,B 0,C 180,E1 -20122.21,E2 -20122.21} C_VEL
LIN {X 0,Y 230.459,Z 730.095,A -85,B 0,C 180,E1 -20124.59,E2 -20124.59} C_VEL
LIN {X 0,Y 229.523,Z 738.071,A -85,B 0,C 180,E1 -20127.077,E2 -20127.077} C_VEL
LIN {X 0,Y 228.901,Z 745.299,A -85,B 0,C 180,E1 -20129.889,E2 -20129.889} C_VEL
LIN {X 0,Y 228.471,Z 750.711,A -85,B 0,C 180,E1 -20132.521,E2 -20132.521} C_VEL
LIN {X 0,Y 228.312,Z 755.363,A -85,B 0,C 180,E1 -20135.445,E2 -20135.445} C_VEL
LIN {X 0,Y 228.555,Z 758.69,A -85,B 0,C 180,E1 -20138.346,E2 -20138.346} C_VEL
LIN {X 0,Y 229.354,Z 761.118,A -85,B 0,C 180,E1 -20141.783,E2 -20141.783} C_VEL
LIN {X 0,Y 230.187,Z 761.874,A -85,B 0,C 180,E1 -20144.051,E2 -20144.051} C_VEL
LIN {X 0,Y 231.337,Z 761.928,A -85,B 0,C 180,E1 -20146.438,E2 -20146.438} C_VEL
LIN {X 0,Y 233.089,Z 760.898,A -85,B 0,C 180,E1 -20149.248,E2 -20149.248} C_VEL
LIN {X 0,Y 233.507,Z 760.225,A -85,B 0,C 180,E1 -20150.686,E2 -20150.686} C_VEL
LIN {X 0,Y 232.717,Z 758.912,A -85,B 0,C 180,E1 -20153.095,E2 -20153.095} C_VEL
LIN {X 0,Y 232.184,Z 756.841,A -85,B 0,C 180,E1 -20155.478,E2 -20155.478} C_VEL
LIN {X 0,Y 232.98,Z 754.983,A -85,B 0,C 180,E1 -20156.843,E2 -20156.843} C_VEL
LIN {X 0,Y 235.745,Z 750.744,A -85,B 0,C 180,E1 -20159.146,E2 -20159.146} C_VEL
LIN {X 0,Y 239.742,Z 743.774,A -85,B 0,C 180,E1 -20161.978,E2 -20161.978} C_VEL
LIN {X 0,Y 243.826,Z 735.414,A -85,B 0,C 180,E1 -20164.546,E2 -20164.546} C_VEL
LIN {X 0,Y 247.691,Z 726.225,A -85,B 0,C 180,E1 -20166.757,E2 -20166.757} C_VEL
LIN {X 0,Y 251.31,Z 716.082,A -85,B 0,C 180,E1 -20168.645,E2 -20168.645} C_VEL
LIN {X 0,Y 254.671,Z 704.71,A -85,B 0,C 180,E1 -20170.333,E2 -20170.333} C_VEL
LIN {X 0,Y 257.259,Z 693.739,A -85,B 0,C 180,E1 -20171.623,E2 -20171.623} C_VEL
LIN {X 0,Y 259.591,Z 681.03,A -85,B 0,C 180,E1 -20172.768,E2 -20172.768} C_VEL
LIN {X 0,Y 260.996,Z 669.226,A -85,B 0,C 180,E1 -20173.588,E2 -20173.588} C_VEL
LIN {X 0,Y 263.187,Z 645.05,A -85,B 0,C 180,E1 -20174.76,E2 -20174.76} C_VEL
LIN {X 0,Y 264.708,Z 630.711,A -85,B 0,C 180,E1 -20175.397,E2 -20175.397} C_VEL
LIN {X 0,Y 260.803,Z 623.225,A -85,B 0,C 180,E1 -20177.615,E2 -20177.615} C_VEL
LIN {X 0,Y 257.486,Z 617.496,A -85,B 0,C 180,E1 -20179.786,E2 -20179.786} C_VEL
LIN {X 0,Y 254.335,Z 612.431,A -85,B 0,C 180,E1 -20182.318,E2 -20182.318} C_VEL
LIN {X 0,Y 252.642,Z 610.676,A -85,B 0,C 180,E1 -20183.887,E2 -20183.887} C_VEL
LIN {X 0,Y 250.215,Z 608.645,A -85,B 0,C 180,E1 -20186.706,E2 -20186.706} C_VEL
LIN {X 0,Y 248.109,Z 608.41,A -85,B 0,C 180,E1 -20190.655,E2 -20190.655} C_VEL
LIN {X 0,Y 247.756,Z 609.054,A -85,B 0,C 180,E1 -20193.25,E2 -20193.25} C_VEL
LIN {X 0,Y 248.242,Z 611.87,A -85,B 0,C 180,E1 -20196.644,E2 -20196.644} C_VEL
LIN {X 0,Y 248.979,Z 614.324,A -85,B 0,C 180,E1 -20198.505,E2 -20198.505} C_VEL
LIN {X 0,Y 251.808,Z 621.838,A -85,B 0,C 180,E1 -20202.554,E2 -20202.554} C_VEL
LIN {X 0,Y 252.843,Z 624.305,A -85,B 0,C 180,E1 -20203.614,E2 -20203.614} C_VEL
LIN {X 0,Y 255.556,Z 631.464,A -85,B 0,C 180,E1 -20206.044,E2 -20206.044} C_VEL
LIN {X 0,Y 257.844,Z 638.006,A -85,B 0,C 180,E1 -20207.819,E2 -20207.819} C_VEL
LIN {X 0,Y 259.24,Z 642.325,A -85,B 0,C 180,E1 -20208.807,E2 -20208.807} C_VEL
LIN {X 0,Y 259.768,Z 658.81,A -85,B 0,C 180,E1 -20210.441,E2 -20210.441} C_VEL
LIN {X 0,Y 259.837,Z 673.524,A -85,B 0,C 180,E1 -20211.62,E2 -20211.62} C_VEL
LIN {X 0,Y 259.295,Z 689.924,A -85,B 0,C 180,E1 -20212.688,E2 -20212.688} C_VEL
LIN {X 0,Y 256.707,Z 712.057,A -85,B 0,C 180,E1 -20213.624,E2 -20213.624} C_VEL
LIN {X 0,Y 254.127,Z 725.368,A -85,B 0,C 180,E1 -20214.39,E2 -20214.39} C_VEL
LIN {X 0,Y 250.758,Z 738.594,A -85,B 0,C 180,E1 -20215.423,E2 -20215.423} C_VEL
LIN {X 0,Y 246.739,Z 751.408,A -85,B 0,C 180,E1 -20216.751,E2 -20216.751} C_VEL
LIN {X 0,Y 242.047,Z 764.178,A -85,B 0,C 180,E1 -20218.493,E2 -20218.493} C_VEL
LIN {X 0,Y 237.67,Z 774.663,A -85,B 0,C 180,E1 -20220.312,E2 -20220.312} C_VEL
LIN {X 0,Y 235.93,Z 778.86,A -85,B 0,C 180,E1 -20221.173,E2 -20221.173} C_VEL
LIN {X 0,Y 233.842,Z 790.406,A -85,B 0,C 180,E1 -20222.48,E2 -20222.48} C_VEL
LIN {X 0,Y 231.427,Z 801.551,A -85,B 0,C 180,E1 -20224.119,E2 -20224.119} C_VEL
LIN {X 0,Y 228.988,Z 811.591,A -85,B 0,C 180,E1 -20226.007,E2 -20226.007} C_VEL
LIN {X 0,Y 226.648,Z 820.638,A -85,B 0,C 180,E1 -20228.157,E2 -20228.157} C_VEL
LIN {X 0,Y 224.256,Z 829.451,A -85,B 0,C 180,E1 -20230.79,E2 -20230.79} C_VEL
LIN {X 0,Y 222.238,Z 836.501,A -85,B 0,C 180,E1 -20233.466,E2 -20233.466} C_VEL
LIN {X 0,Y 220.624,Z 842.106,A -85,B 0,C 180,E1 -20236.179,E2 -20236.179} C_VEL
LIN {X 0,Y 219.621,Z 846.508,A -85,B 0,C 180,E1 -20238.932,E2 -20238.932} C_VEL
LIN {X 0,Y 219.141,Z 848.828,A -85,B 0,C 180,E1 -20240.774,E2 -20240.774} C_VEL
LIN {X 0,Y 218.797,Z 850.718,A -85,B 0,C 180,E1 -20242.62,E2 -20242.62} C_VEL
LIN {X 0,Y 218.625,Z 852.612,A -85,B 0,C 180,E1 -20245.232,E2 -20245.232} C_VEL
LIN {X 0,Y 218.663,Z 853.769,A -85,B 0,C 180,E1 -20248.16,E2 -20248.16} C_VEL
LIN {X 0,Y 218.742,Z 853.987,A -85,B 0,C 180,E1 -20250.002,E2 -20250.002} C_VEL
LIN {X 0,Y 218.654,Z 853.757,A -85,B 0,C 180,E1 -20251.843,E2 -20251.843} C_VEL
LIN {X 0,Y 218.659,Z 852.521,A -85,B 0,C 180,E1 -20254.875,E2 -20254.875} C_VEL
LIN {X 0,Y 218.803,Z 850.674,A -85,B 0,C 180,E1 -20257.383,E2 -20257.383} C_VEL
LIN {X 0,Y 219.357,Z 847.688,A -85,B 0,C 180,E1 -20260.151,E2 -20260.151} C_VEL
LIN {X 0,Y 220.22,Z 843.639,A -85,B 0,C 180,E1 -20262.91,E2 -20262.91} C_VEL
LIN {X 0,Y 221.896,Z 837.401,A -85,B 0,C 180,E1 -20266.091,E2 -20266.091} C_VEL
LIN {X 0,Y 223.832,Z 830.601,A -85,B 0,C 180,E1 -20268.775,E2 -20268.775} C_VEL
LIN {X 0,Y 225.926,Z 823.026,A -85,B 0,C 180,E1 -20271.163,E2 -20271.163} C_VEL
LIN {X 0,Y 227.916,Z 815.267,A -85,B 0,C 180,E1 -20273.152,E2 -20273.152} C_VEL
LIN {X 0,Y 230.592,Z 804.886,A -85,B 0,C 180,E1 -20275.259,E2 -20275.259} C_VEL
LIN {X 0,Y 233.224,Z 793.19,A -85,B 0,C 180,E1 -20277.116,E2 -20277.116} C_VEL
LIN {X 0,Y 235.372,Z 781.389,A -85,B 0,C 180,E1 -20278.539,E2 -20278.539} C_VEL
LIN {X 0,Y 237.26,Z 769.147,A -85,B 0,C 180,E1 -20279.625,E2 -20279.625} C_VEL
LIN {X 0,Y 238.783,Z 756.94,A -85,B 0,C 180,E1 -20280.364,E2 -20280.364} C_VEL
LIN {X 0,Y 239.62,Z 743.632,A -85,B 0,C 180,E1 -20280.871,E2 -20280.871} C_VEL
LIN {X 0,Y 241.609,Z 688.038,A -85,B 0,C 180,E1 -20282.482,E2 -20282.482} C_VEL
LIN {X 0,Y 239.31,Z 661.402,A -85,B 0,C 180,E1 -20283.764,E2 -20283.764} C_VEL
LIN {X 0,Y 236.01,Z 635.107,A -85,B 0,C 180,E1 -20285.249,E2 -20285.249} C_VEL
LIN {X 0,Y 235.888,Z 632.522,A -85,B 0,C 180,E1 -20285.522,E2 -20285.522} C_VEL
LIN {X 0,Y 236.104,Z 617.065,A -85,B 0,C 180,E1 -20287.516,E2 -20287.516} C_VEL
LIN {X 0,Y 232.292,Z 603.013,A -85,B 0,C 180,E1 -20290.138,E2 -20290.138} C_VEL
LIN {X 0,Y 229.54,Z 593.532,A -85,B 0,C 180,E1 -20292.123,E2 -20292.123} C_VEL
LIN {X 0,Y 226.724,Z 584.408,A -85,B 0,C 180,E1 -20294.161,E2 -20294.161} C_VEL
LIN {X 0,Y 225.884,Z 582.466,A -85,B 0,C 180,E1 -20294.703,E2 -20294.703} C_VEL
LIN {X 0,Y 222.304,Z 576.548,A -85,B 0,C 180,E1 -20296.647,E2 -20296.647} C_VEL
LIN {X 0,Y 221.168,Z 574.545,A -85,B 0,C 180,E1 -20297.311,E2 -20297.311} C_VEL
LIN {X 0,Y 220.788,Z 572.967,A -85,B 0,C 180,E1 -20297.741,E2 -20297.741} C_VEL
LIN {X 0,Y 220.809,Z 572.981,A -85,B 0,C 180,E1 -20300.464,E2 -20300.464} C_VEL
LIN {X 0,Y 220.803,Z 572.972,A -85,B 0,C 180,E1 -20305.045,E2 -20305.045} C_VEL
LIN {X 0,Y 220.871,Z 572.948,A -85,B 0,C 180,E1 -20309.395,E2 -20309.395} C_VEL
LIN {X 0,Y 220.898,Z 572.954,A -85,B 0,C 180,E1 -20313.55,E2 -20313.55} C_VEL
LIN {X 0,Y 220.868,Z 572.965,A -85,B 0,C 180,E1 -20317.552,E2 -20317.552} C_VEL
LIN {X 0,Y 220.987,Z 572.926,A -85,B 0,C 180,E1 -20322.572,E2 -20322.572} C_VEL
LIN {X 0,Y 221.013,Z 572.944,A -85,B 0,C 180,E1 -20327.139,E2 -20327.139} C_VEL
LIN {X 0,Y 221.207,Z 572.903,A -85,B 0,C 180,E1 -20330.86,E2 -20330.86} C_VEL
LIN {X 0,Y 221.262,Z 572.922,A -85,B 0,C 180,E1 -20332.701,E2 -20332.701} C_VEL
LIN {X 0,Y 221.514,Z 572.86,A -85,B 0,C 180,E1 -20338.182,E2 -20338.182} C_VEL
LIN {X 0,Y 221.514,Z 572.89,A -85,B 0,C 180,E1 -20341.818,E2 -20341.818} C_VEL
LIN {X 0,Y 221.292,Z 572.907,A -85,B 0,C 180,E1 -20347.298,E2 -20347.298} C_VEL
LIN {X 0,Y 221.11,Z 572.919,A -85,B 0,C 180,E1 -20350.994,E2 -20350.994} C_VEL
LIN {X 0,Y 221.019,Z 572.952,A -85,B 0,C 180,E1 -20356.63,E2 -20356.63} C_VEL
LIN {X 0,Y 220.896,Z 572.948,A -85,B 0,C 180,E1 -20360.486,E2 -20360.486} C_VEL
LIN {X 0,Y 220.871,Z 572.953,A -85,B 0,C 180,E1 -20364.435,E2 -20364.435} C_VEL
LIN {X 0,Y 220.84,Z 572.976,A -85,B 0,C 180,E1 -20368.513,E2 -20368.513} C_VEL
LIN {X 0,Y 220.821,Z 572.977,A -85,B 0,C 180,E1 -20372.756,E2 -20372.756} C_VEL
LIN {X 0,Y 220.894,Z 573.092,A -85,B 0,C 180,E1 -20376.695,E2 -20376.695} C_VEL
LIN {X 0,Y 221.482,Z 575.17,A -85,B 0,C 180,E1 -20377.504,E2 -20377.504} C_VEL
LIN {X 0,Y 223.815,Z 580.032,A -85,B 0,C 180,E1 -20379.649,E2 -20379.649} C_VEL
LIN {X 0,Y 227.017,Z 588.251,A -85,B 0,C 180,E1 -20382.928,E2 -20382.928} C_VEL
LIN {X 0,Y 230.887,Z 599.466,A -85,B 0,C 180,E1 -20386.932,E2 -20386.932} C_VEL
LIN {X 0,Y 234.224,Z 611.291,A -85,B 0,C 180,E1 -20390.656,E2 -20390.656} C_VEL
LIN {X 0,Y 236.839,Z 623.017,A -85,B 0,C 180,E1 -20393.96,E2 -20393.96} C_VEL
LIN {X 0,Y 237.544,Z 626.89,A -85,B 0,C 180,E1 -20394.897,E2 -20394.897} C_VEL
LIN {X 0,Y 242.127,Z 657.244,A -85,B 0,C 180,E1 -20396.724,E2 -20396.724} C_VEL
LIN {X 0,Y 243.073,Z 666.209,A -85,B 0,C 180,E1 -20397.182,E2 -20397.182} C_VEL
LIN {X 0,Y 240.034,Z 739.185,A -85,B 0,C 180,E1 -20399.298,E2 -20399.298} C_VEL
LIN {X 0,Y 238.894,Z 752.467,A -85,B 0,C 180,E1 -20399.991,E2 -20399.991} C_VEL
LIN {X 0,Y 237.262,Z 764.995,A -85,B 0,C 180,E1 -20400.983,E2 -20400.983} C_VEL
LIN {X 0,Y 235.432,Z 776.23,A -85,B 0,C 180,E1 -20402.196,E2 -20402.196} C_VEL
LIN {X 0,Y 233.013,Z 787.839,A -85,B 0,C 180,E1 -20403.824,E2 -20403.824} C_VEL
LIN {X 0,Y 230.603,Z 798.19,A -85,B 0,C 180,E1 -20405.704,E2 -20405.704} C_VEL
LIN {X 0,Y 228.201,Z 808.089,A -85,B 0,C 180,E1 -20407.99,E2 -20407.99} C_VEL
LIN {X 0,Y 225.752,Z 816.522,A -85,B 0,C 180,E1 -20410.447,E2 -20410.447} C_VEL
LIN {X 0,Y 223.562,Z 823.74,A -85,B 0,C 180,E1 -20413.094,E2 -20413.094} C_VEL
LIN {X 0,Y 221.583,Z 830.359,A -85,B 0,C 180,E1 -20416.237,E2 -20416.237} C_VEL
LIN {X 0,Y 220.343,Z 834.698,A -85,B 0,C 180,E1 -20418.966,E2 -20418.966} C_VEL
LIN {X 0,Y 219.747,Z 836.979,A -85,B 0,C 180,E1 -20420.797,E2 -20420.797} C_VEL
LIN {X 0,Y 219.009,Z 840.045,A -85,B 0,C 180,E1 -20424.152,E2 -20424.152} C_VEL
LIN {X 0,Y 218.742,Z 841.249,A -85,B 0,C 180,E1 -20426.314,E2 -20426.314} C_VEL
LIN {X 0,Y 218.666,Z 841.86,A -85,B 0,C 180,E1 -20428.157,E2 -20428.157} C_VEL
LIN {X 0,Y 218.661,Z 842.091,A -85,B 0,C 180,E1 -20429.998,E2 -20429.998} C_VEL
LIN {X 0,Y 218.664,Z 841.895,A -85,B 0,C 180,E1 -20431.84,E2 -20431.84} C_VEL
LIN {X 0,Y 218.955,Z 840.338,A -85,B 0,C 180,E1 -20435.524,E2 -20435.524} C_VEL
LIN {X 0,Y 219.273,Z 838.967,A -85,B 0,C 180,E1 -20437.364,E2 -20437.364} C_VEL
LIN {X 0,Y 219.988,Z 836.086,A -85,B 0,C 180,E1 -20440.118,E2 -20440.118} C_VEL
LIN {X 0,Y 221.082,Z 832.167,A -85,B 0,C 180,E1 -20442.856,E2 -20442.856} C_VEL
LIN {X 0,Y 222.627,Z 827.088,A -85,B 0,C 180,E1 -20445.563,E2 -20445.563} C_VEL
LIN {X 0,Y 224.538,Z 820.686,A -85,B 0,C 180,E1 -20448.238,E2 -20448.238} C_VEL
LIN {X 0,Y 226.984,Z 812.712,A -85,B 0,C 180,E1 -20450.857,E2 -20450.857} C_VEL
LIN {X 0,Y 229.256,Z 804.128,A -85,B 0,C 180,E1 -20453.121,E2 -20453.121} C_VEL
LIN {X 0,Y 231.568,Z 794.515,A -85,B 0,C 180,E1 -20455.142,E2 -20455.142} C_VEL
LIN {X 0,Y 233.842,Z 784.6,A -85,B 0,C 180,E1 -20456.794,E2 -20456.794} C_VEL
LIN {X 0,Y 235.956,Z 773.812,A -85,B 0,C 180,E1 -20458.217,E2 -20458.217} C_VEL
LIN {X 0,Y 237.823,Z 761.889,A -85,B 0,C 180,E1 -20459.423,E2 -20459.423} C_VEL
LIN {X 0,Y 239.255,Z 749.495,A -85,B 0,C 180,E1 -20460.321,E2 -20460.321} C_VEL
LIN {X 0,Y 240.246,Z 736.942,A -85,B 0,C 180,E1 -20460.913,E2 -20460.913} C_VEL
LIN {X 0,Y 243.025,Z 667.578,A -85,B 0,C 180,E1 -20462.917,E2 -20462.917} C_VEL
LIN {X 0,Y 238.999,Z 642.034,A -85,B 0,C 180,E1 -20464.455,E2 -20464.455} C_VEL
LIN {X 0,Y 236.303,Z 627.119,A -85,B 0,C 180,E1 -20465.485,E2 -20465.485} C_VEL
LIN {X 0,Y 236.23,Z 624.306,A -85,B 0,C 180,E1 -20466.222,E2 -20466.222} C_VEL
LIN {X 0,Y 234.262,Z 614.224,A -85,B 0,C 180,E1 -20469.294,E2 -20469.294} C_VEL
LIN {X 0,Y 233.455,Z 610.774,A -85,B 0,C 180,E1 -20470.401,E2 -20470.401} C_VEL
LIN {X 0,Y 232.608,Z 609.466,A -85,B 0,C 180,E1 -20470.944,E2 -20470.944} C_VEL
LIN {X 0,Y 231.341,Z 608.472,A -85,B 0,C 180,E1 -20471.506,E2 -20471.506} C_VEL
LIN {X 0,Y 230.053,Z 645.935,A -85,B 0,C 180,E1 -20473.106,E2 -20473.106} C_VEL
LIN {X 0,Y 229.678,Z 661.055,A -85,B 0,C 180,E1 -20473.87,E2 -20473.87} C_VEL
LIN {X 0,Y 228.992,Z 674.477,A -85,B 0,C 180,E1 -20474.899,E2 -20474.899} C_VEL
LIN {X 0,Y 228.048,Z 687.505,A -85,B 0,C 180,E1 -20476.252,E2 -20476.252} C_VEL
LIN {X 0,Y 226.856,Z 700.491,A -85,B 0,C 180,E1 -20478.029,E2 -20478.029} C_VEL
LIN {X 0,Y 225.614,Z 712.016,A -85,B 0,C 180,E1 -20480.023,E2 -20480.023} C_VEL
LIN {X 0,Y 224.359,Z 722.787,A -85,B 0,C 180,E1 -20482.35,E2 -20482.35} C_VEL
LIN {X 0,Y 223.242,Z 732.418,A -85,B 0,C 180,E1 -20484.933,E2 -20484.933} C_VEL
LIN {X 0,Y 222.312,Z 740.137,A -85,B 0,C 180,E1 -20487.491,E2 -20487.491} C_VEL
LIN {X 0,Y 221.696,Z 747.57,A -85,B 0,C 180,E1 -20490.569,E2 -20490.569} C_VEL
LIN {X 0,Y 221.316,Z 753.233,A -85,B 0,C 180,E1 -20493.604,E2 -20493.604} C_VEL
LIN {X 0,Y 221.321,Z 758.032,A -85,B 0,C 180,E1 -20497.05,E2 -20497.05} C_VEL
LIN {X 0,Y 221.742,Z 760.514,A -85,B 0,C 180,E1 -20499.596,E2 -20499.596} C_VEL
LIN {X 0,Y 222.236,Z 761.895,A -85,B 0,C 180,E1 -20501.564,E2 -20501.564} C_VEL
LIN {X 0,Y 222.94,Z 762.74,A -85,B 0,C 180,E1 -20503.518,E2 -20503.518} C_VEL
LIN {X 0,Y 224.22,Z 763.149,A -85,B 0,C 180,E1 -20506.319,E2 -20506.319} C_VEL
LIN {X 0,Y 226.273,Z 762.302,A -85,B 0,C 180,E1 -20509.592,E2 -20509.592} C_VEL
LIN {X 0,Y 227.542,Z 761.397,A -85,B 0,C 180,E1 -20511.239,E2 -20511.239} C_VEL
LIN {X 0,Y 229.797,Z 759.055,A -85,B 0,C 180,E1 -20513.855,E2 -20513.855} C_VEL
LIN {X 0,Y 232.98,Z 754.983,A -85,B 0,C 180,E1 -20516.843,E2 -20516.843} C_VEL
LIN {X 0,Y 233.877,Z 752.95,A -85,B 0,C 180,E1 -20518.19,E2 -20518.19} C_VEL
LIN {X 0,Y 233.972,Z 749.641,A -85,B 0,C 180,E1 -20520.488,E2 -20520.488} C_VEL
LIN {X 0,Y 234.358,Z 745.731,A -85,B 0,C 180,E1 -20522.703,E2 -20522.703} C_VEL
LIN {X 0,Y 235.646,Z 742.698,A -85,B 0,C 180,E1 -20523.89,E2 -20523.89} C_VEL
LIN {X 0,Y 239.772,Z 734.431,A -85,B 0,C 180,E1 -20526.31,E2 -20526.31} C_VEL
LIN {X 0,Y 243.486,Z 725.753,A -85,B 0,C 180,E1 -20528.298,E2 -20528.298} C_VEL
LIN {X 0,Y 247.437,Z 715.187,A -85,B 0,C 180,E1 -20530.225,E2 -20530.225} C_VEL
LIN {X 0,Y 250.619,Z 704.715,A -85,B 0,C 180,E1 -20531.731,E2 -20531.731} C_VEL
LIN {X 0,Y 253.281,Z 693.765,A -85,B 0,C 180,E1 -20532.988,E2 -20532.988} C_VEL
LIN {X 0,Y 255.751,Z 680.292,A -85,B 0,C 180,E1 -20534.193,E2 -20534.193} C_VEL
LIN {X 0,Y 257.377,Z 667.3,A -85,B 0,C 180,E1 -20535.029,E2 -20535.029} C_VEL
LIN {X 0,Y 259.578,Z 645.086,A -85,B 0,C 180,E1 -20536.109,E2 -20536.109} C_VEL
LIN {X 0,Y 260.723,Z 634.399,A -85,B 0,C 180,E1 -20536.607,E2 -20536.607} C_VEL
LIN {X 0,Y 257.336,Z 627.735,A -85,B 0,C 180,E1 -20538.769,E2 -20538.769} C_VEL
LIN {X 0,Y 254.779,Z 622.999,A -85,B 0,C 180,E1 -20540.66,E2 -20540.66} C_VEL
LIN {X 0,Y 252.3,Z 618.948,A -85,B 0,C 180,E1 -20542.799,E2 -20542.799} C_VEL
LIN {X 0,Y 250.847,Z 617.426,A -85,B 0,C 180,E1 -20544.208,E2 -20544.208} C_VEL
LIN {X 0,Y 248.645,Z 615.565,A -85,B 0,C 180,E1 -20546.888,E2 -20546.888} C_VEL
LIN {X 0,Y 246.586,Z 615.445,A -85,B 0,C 180,E1 -20551.24,E2 -20551.24} C_VEL
LIN {X 0,Y 246.331,Z 616.078,A -85,B 0,C 180,E1 -20553.246,E2 -20553.246} C_VEL
LIN {X 0,Y 246.826,Z 619.061,A -85,B 0,C 180,E1 -20556.723,E2 -20556.723} C_VEL
LIN {X 0,Y 247.873,Z 623.08,A -85,B 0,C 180,E1 -20559.335,E2 -20559.335} C_VEL
LIN {X 0,Y 250.439,Z 629.883,A -85,B 0,C 180,E1 -20562.77,E2 -20562.77} C_VEL
LIN {X 0,Y 252.979,Z 637.323,A -85,B 0,C 180,E1 -20565.343,E2 -20565.343} C_VEL
LIN {X 0,Y 255.083,Z 644.008,A -85,B 0,C 180,E1 -20567.167,E2 -20567.167} C_VEL
LIN {X 0,Y 255.772,Z 646.375,A -85,B 0,C 180,E1 -20567.715,E2 -20567.715} C_VEL
LIN {X 0,Y 256.051,Z 661.867,A -85,B 0,C 180,E1 -20569.271,E2 -20569.271} C_VEL
LIN {X 0,Y 255.819,Z 676.617,A -85,B 0,C 180,E1 -20570.468,E2 -20570.468} C_VEL
LIN {X 0,Y 255.194,Z 691.911,A -85,B 0,C 180,E1 -20571.471,E2 -20571.471} C_VEL
LIN {X 0,Y 252.687,Z 711.006,A -85,B 0,C 180,E1 -20572.276,E2 -20572.276} C_VEL
LIN {X 0,Y 249.64,Z 725.445,A -85,B 0,C 180,E1 -20573.132,E2 -20573.132} C_VEL
LIN {X 0,Y 246.128,Z 738.337,A -85,B 0,C 180,E1 -20574.174,E2 -20574.174} C_VEL
LIN {X 0,Y 241.934,Z 750.916,A -85,B 0,C 180,E1 -20575.499,E2 -20575.499} C_VEL
LIN {X 0,Y 237.498,Z 762.392,A -85,B 0,C 180,E1 -20577.063,E2 -20577.063} C_VEL
LIN {X 0,Y 233.374,Z 771.915,A -85,B 0,C 180,E1 -20578.705,E2 -20578.705} C_VEL
LIN {X 0,Y 229.388,Z 780.648,A -85,B 0,C 180,E1 -20580.522,E2 -20580.522} C_VEL
LIN {X 0,Y 227.25,Z 791.793,A -85,B 0,C 180,E1 -20581.862,E2 -20581.862} C_VEL
LIN {X 0,Y 224.755,Z 802.614,A -85,B 0,C 180,E1 -20583.541,E2 -20583.541} C_VEL
LIN {X 0,Y 221.977,Z 813.344,A -85,B 0,C 180,E1 -20585.697,E2 -20585.697} C_VEL
LIN {X 0,Y 219.459,Z 822.455,A -85,B 0,C 180,E1 -20588.016,E2 -20588.016} C_VEL
LIN {X 0,Y 217.136,Z 830.544,A -85,B 0,C 180,E1 -20590.626,E2 -20590.626} C_VEL
LIN {X 0,Y 215.084,Z 837.315,A -85,B 0,C 180,E1 -20593.389,E2 -20593.389} C_VEL
LIN {X 0,Y 213.288,Z 843.526,A -85,B 0,C 180,E1 -20596.666,E2 -20596.666} C_VEL
LIN {X 0,Y 212.352,Z 847.556,A -85,B 0,C 180,E1 -20599.514,E2 -20599.514} C_VEL
LIN {X 0,Y 211.726,Z 850.525,A -85,B 0,C 180,E1 -20602.372,E2 -20602.372} C_VEL
LIN {X 0,Y 211.542,Z 852.574,A -85,B 0,C 180,E1 -20605.333,E2 -20605.333} C_VEL
LIN {X 0,Y 211.558,Z 853.576,A -85,B 0,C 180,E1 -20608.098,E2 -20608.098} C_VEL
LIN {X 0,Y 211.654,Z 853.794,A -85,B 0,C 180,E1 -20610.002,E2 -20610.002} C_VEL
LIN {X 0,Y 211.55,Z 853.563,A -85,B 0,C 180,E1 -20611.905,E2 -20611.905} C_VEL
LIN {X 0,Y 211.543,Z 852.545,A -85,B 0,C 180,E1 -20614.671,E2 -20614.671} C_VEL
LIN {X 0,Y 211.733,Z 850.479,A -85,B 0,C 180,E1 -20617.631,E2 -20617.631} C_VEL
LIN {X 0,Y 212.354,Z 847.494,A -85,B 0,C 180,E1 -20620.489,E2 -20620.489} C_VEL
LIN {X 0,Y 213.253,Z 843.444,A -85,B 0,C 180,E1 -20623.339,E2 -20623.339} C_VEL
LIN {X 0,Y 215.062,Z 837.208,A -85,B 0,C 180,E1 -20626.616,E2 -20626.616} C_VEL
LIN {X 0,Y 217.113,Z 830.409,A -85,B 0,C 180,E1 -20629.379,E2 -20629.379} C_VEL
LIN {X 0,Y 219.194,Z 823.167,A -85,B 0,C 180,E1 -20631.737,E2 -20631.737} C_VEL
LIN {X 0,Y 221.376,Z 815.077,A -85,B 0,C 180,E1 -20633.878,E2 -20633.878} C_VEL
LIN {X 0,Y 224.167,Z 804.698,A -85,B 0,C 180,E1 -20636.036,E2 -20636.036} C_VEL
LIN {X 0,Y 226.616,Z 794.423,A -85,B 0,C 180,E1 -20637.724,E2 -20637.724} C_VEL
LIN {X 0,Y 228.84,Z 783.146,A -85,B 0,C 180,E1 -20639.18,E2 -20639.18} C_VEL
LIN {X 0,Y 230.962,Z 770.246,A -85,B 0,C 180,E1 -20640.391,E2 -20640.391} C_VEL
LIN {X 0,Y 232.586,Z 757.73,A -85,B 0,C 180,E1 -20641.198,E2 -20641.198} C_VEL
LIN {X 0,Y 233.541,Z 744.112,A -85,B 0,C 180,E1 -20641.745,E2 -20641.745} C_VEL
LIN {X 0,Y 235.639,Z 689.001,A -85,B 0,C 180,E1 -20643.373,E2 -20643.373} C_VEL
LIN {X 0,Y 233.538,Z 663.445,A -85,B 0,C 180,E1 -20644.638,E2 -20644.638} C_VEL
LIN {X 0,Y 230.466,Z 638.152,A -85,B 0,C 180,E1 -20646.111,E2 -20646.111} C_VEL
LIN {X 0,Y 229.872,Z 633.5,A -85,B 0,C 180,E1 -20646.438,E2 -20646.438} C_VEL
LIN {X 0,Y 230.278,Z 619.735,A -85,B 0,C 180,E1 -20648.28,E2 -20648.28} C_VEL
LIN {X 0,Y 227.058,Z 607.385,A -85,B 0,C 180,E1 -20650.681,E2 -20650.681} C_VEL
LIN {X 0,Y 224.138,Z 596.981,A -85,B 0,C 180,E1 -20652.922,E2 -20652.922} C_VEL
LIN {X 0,Y 222.108,Z 589.654,A -85,B 0,C 180,E1 -20654.605,E2 -20654.605} C_VEL
LIN {X 0,Y 220.624,Z 586.546,A -85,B 0,C 180,E1 -20655.508,E2 -20655.508} C_VEL
LIN {X 0,Y 216.189,Z 578.364,A -85,B 0,C 180,E1 -20658.209,E2 -20658.209} C_VEL
LIN {X 0,Y 214.22,Z 575.7,A -85,B 0,C 180,E1 -20659.409,E2 -20659.409} C_VEL
LIN {X 0,Y 213.759,Z 573.851,A -85,B 0,C 180,E1 -20660.022,E2 -20660.022} C_VEL
LIN {X 0,Y 213.774,Z 573.85,A -85,B 0,C 180,E1 -20665.276,E2 -20665.276} C_VEL
LIN {X 0,Y 213.784,Z 573.83,A -85,B 0,C 180,E1 -20668.732,E2 -20668.732} C_VEL
LIN {X 0,Y 213.829,Z 573.847,A -85,B 0,C 180,E1 -20672.604,E2 -20672.604} C_VEL
LIN {X 0,Y 213.822,Z 573.833,A -85,B 0,C 180,E1 -20676.974,E2 -20676.974} C_VEL
LIN {X 0,Y 213.946,Z 573.803,A -85,B 0,C 180,E1 -20682.804,E2 -20682.804} C_VEL
LIN {X 0,Y 213.954,Z 573.829,A -85,B 0,C 180,E1 -20686.707,E2 -20686.707} C_VEL
LIN {X 0,Y 214.145,Z 573.779,A -85,B 0,C 180,E1 -20690.555,E2 -20690.555} C_VEL
LIN {X 0,Y 214.103,Z 573.812,A -85,B 0,C 180,E1 -20694.349,E2 -20694.349} C_VEL
LIN {X 0,Y 214.447,Z 573.739,A -85,B 0,C 180,E1 -20698.122,E2 -20698.122} C_VEL
LIN {X 0,Y 214.549,Z 573.751,A -85,B 0,C 180,E1 -20700,E2 -20700} C_VEL
LIN {X 0,Y 214.448,Z 573.77,A -85,B 0,C 180,E1 -20701.878,E2 -20701.878} C_VEL
LIN {X 0,Y 214.23,Z 573.79,A -85,B 0,C 180,E1 -20707.54,E2 -20707.54} C_VEL
LIN {X 0,Y 214.026,Z 573.797,A -85,B 0,C 180,E1 -20711.363,E2 -20711.363} C_VEL
LIN {X 0,Y 213.936,Z 573.834,A -85,B 0,C 180,E1 -20715.237,E2 -20715.237} C_VEL
LIN {X 0,Y 213.843,Z 573.82,A -85,B 0,C 180,E1 -20719.187,E2 -20719.187} C_VEL
LIN {X 0,Y 213.851,Z 573.841,A -85,B 0,C 180,E1 -20723.227,E2 -20723.227} C_VEL
LIN {X 0,Y 213.833,Z 573.843,A -85,B 0,C 180,E1 -20727.45,E2 -20727.45} C_VEL
LIN {X 0,Y 213.772,Z 573.842,A -85,B 0,C 180,E1 -20731.737,E2 -20731.737} C_VEL
LIN {X 0,Y 213.794,Z 573.95,A -85,B 0,C 180,E1 -20734.55,E2 -20734.55} C_VEL
LIN {X 0,Y 215.033,Z 577.047,A -85,B 0,C 180,E1 -20736.037,E2 -20736.037} C_VEL
LIN {X 0,Y 218.426,Z 584.621,A -85,B 0,C 180,E1 -20739.446,E2 -20739.446} C_VEL
LIN {X 0,Y 221.413,Z 592.44,A -85,B 0,C 180,E1 -20742.645,E2 -20742.645} C_VEL
LIN {X 0,Y 225.09,Z 603.37,A -85,B 0,C 180,E1 -20746.613,E2 -20746.613} C_VEL
LIN {X 0,Y 228.25,Z 614.857,A -85,B 0,C 180,E1 -20750.334,E2 -20750.334} C_VEL
LIN {X 0,Y 230.916,Z 626.974,A -85,B 0,C 180,E1 -20753.731,E2 -20753.731} C_VEL
LIN {X 0,Y 232.145,Z 630.505,A -85,B 0,C 180,E1 -20754.087,E2 -20754.087} C_VEL
LIN {X 0,Y 236.498,Z 660.682,A -85,B 0,C 180,E1 -20755.946,E2 -20755.946} C_VEL
LIN {X 0,Y 237.115,Z 667.493,A -85,B 0,C 180,E1 -20756.291,E2 -20756.291} C_VEL
LIN {X 0,Y 233.965,Z 739.318,A -85,B 0,C 180,E1 -20758.411,E2 -20758.411} C_VEL
LIN {X 0,Y 232.779,Z 752.631,A -85,B 0,C 180,E1 -20759.118,E2 -20759.118} C_VEL
LIN {X 0,Y 231.088,Z 765.169,A -85,B 0,C 180,E1 -20760.131,E2 -20760.131} C_VEL
LIN {X 0,Y 229.196,Z 776.41,A -85,B 0,C 180,E1 -20761.371,E2 -20761.371} C_VEL
LIN {X 0,Y 226.97,Z 786.745,A -85,B 0,C 180,E1 -20762.823,E2 -20762.823} C_VEL
LIN {X 0,Y 224.413,Z 797.338,A -85,B 0,C 180,E1 -20764.741,E2 -20764.741} C_VEL
LIN {X 0,Y 221.73,Z 807.725,A -85,B 0,C 180,E1 -20767.152,E2 -20767.152} C_VEL
LIN {X 0,Y 219.522,Z 815.376,A -85,B 0,C 180,E1 -20769.379,E2 -20769.379} C_VEL
LIN {X 0,Y 217.134,Z 822.839,A -85,B 0,C 180,E1 -20772.091,E2 -20772.091} C_VEL
LIN {X 0,Y 215.255,Z 828.828,A -85,B 0,C 180,E1 -20774.858,E2 -20774.858} C_VEL
LIN {X 0,Y 213.757,Z 833.56,A -85,B 0,C 180,E1 -20777.659,E2 -20777.659} C_VEL
LIN {X 0,Y 212.722,Z 837.173,A -85,B 0,C 180,E1 -20780.49,E2 -20780.49} C_VEL
LIN {X 0,Y 212.24,Z 839.032,A -85,B 0,C 180,E1 -20782.387,E2 -20782.387} C_VEL
LIN {X 0,Y 211.893,Z 840.449,A -85,B 0,C 180,E1 -20784.288,E2 -20784.288} C_VEL
LIN {X 0,Y 211.587,Z 842.053,A -85,B 0,C 180,E1 -20788.095,E2 -20788.095} C_VEL
LIN {X 0,Y 211.578,Z 842.283,A -85,B 0,C 180,E1 -20789.998,E2 -20789.998} C_VEL
LIN {X 0,Y 211.566,Z 842.088,A -85,B 0,C 180,E1 -20791.902,E2 -20791.902} C_VEL
LIN {X 0,Y 211.892,Z 840.53,A -85,B 0,C 180,E1 -20795.709,E2 -20795.709} C_VEL
LIN {X 0,Y 212.236,Z 839.159,A -85,B 0,C 180,E1 -20797.61,E2 -20797.61} C_VEL
LIN {X 0,Y 212.996,Z 836.278,A -85,B 0,C 180,E1 -20800.454,E2 -20800.454} C_VEL
LIN {X 0,Y 214.161,Z 832.358,A -85,B 0,C 180,E1 -20803.278,E2 -20803.278} C_VEL
LIN {X 0,Y 215.768,Z 827.279,A -85,B 0,C 180,E1 -20806.071,E2 -20806.071} C_VEL
LIN {X 0,Y 217.807,Z 820.874,A -85,B 0,C 180,E1 -20808.823,E2 -20808.823} C_VEL
LIN {X 0,Y 220.37,Z 812.898,A -85,B 0,C 180,E1 -20811.514,E2 -20811.514} C_VEL
LIN {X 0,Y 222.606,Z 804.819,A -85,B 0,C 180,E1 -20813.712,E2 -20813.712} C_VEL
LIN {X 0,Y 224.906,Z 795.83,A -85,B 0,C 180,E1 -20815.693,E2 -20815.693} C_VEL
LIN {X 0,Y 227.533,Z 784.776,A -85,B 0,C 180,E1 -20817.599,E2 -20817.599} C_VEL
LIN {X 0,Y 229.716,Z 773.981,A -85,B 0,C 180,E1 -20819.055,E2 -20819.055} C_VEL
LIN {X 0,Y 231.679,Z 762.045,A -85,B 0,C 180,E1 -20820.284,E2 -20820.284} C_VEL
LIN {X 0,Y 233.177,Z 749.632,A -85,B 0,C 180,E1 -20821.198,E2 -20821.198} C_VEL
LIN {X 0,Y 234.194,Z 737.035,A -85,B 0,C 180,E1 -20821.803,E2 -20821.803} C_VEL
LIN {X 0,Y 237.057,Z 668.419,A -85,B 0,C 180,E1 -20823.827,E2 -20823.827} C_VEL
LIN {X 0,Y 232.596,Z 639.931,A -85,B 0,C 180,E1 -20825.625,E2 -20825.625} C_VEL
LIN {X 0,Y 230.197,Z 627.961,A -85,B 0,C 180,E1 -20826.511,E2 -20826.511} C_VEL
LIN {X 0,Y 229.954,Z 627.048,A -85,B 0,C 180,E1 -20826.69,E2 -20826.69} C_VEL
LIN {X 0,Y 228.115,Z 617.5,A -85,B 0,C 180,E1 -20829.626,E2 -20829.626} C_VEL
LIN {X 0,Y 226.368,Z 615.831,A -85,B 0,C 180,E1 -20830.48,E2 -20830.48} C_VEL
LIN {X 0,Y 224.28,Z 614.858,A -85,B 0,C 180,E1 -20831.231,E2 -20831.231} C_VEL
LIN {X 0,Y 224.17,Z 614.75,A -85,B 0,C 180,E1 -20831.311,E2 -20831.311} C_VEL
LIN {X 0,Y 222.965,Z 656.452,A -85,B 0,C 180,E1 -20833.163,E2 -20833.163} C_VEL
LIN {X 0,Y 222.292,Z 671.164,A -85,B 0,C 180,E1 -20834.178,E2 -20834.178} C_VEL
LIN {X 0,Y 221.476,Z 683.791,A -85,B 0,C 180,E1 -20835.405,E2 -20835.405} C_VEL
LIN {X 0,Y 220.3,Z 696.908,A -85,B 0,C 180,E1 -20837.085,E2 -20837.085} C_VEL
LIN {X 0,Y 219.133,Z 708.026,A -85,B 0,C 180,E1 -20838.892,E2 -20838.892} C_VEL
LIN {X 0,Y 217.854,Z 719.067,A -85,B 0,C 180,E1 -20841.136,E2 -20841.136} C_VEL
LIN {X 0,Y 216.636,Z 729.265,A -85,B 0,C 180,E1 -20843.697,E2 -20843.697} C_VEL
LIN {X 0,Y 215.586,Z 737.761,A -85,B 0,C 180,E1 -20846.345,E2 -20846.345} C_VEL
LIN {X 0,Y 214.905,Z 744.715,A -85,B 0,C 180,E1 -20848.998,E2 -20848.998} C_VEL
LIN {X 0,Y 214.449,Z 750.135,A -85,B 0,C 180,E1 -20851.519,E2 -20851.519} C_VEL
LIN {X 0,Y 214.166,Z 755.664,A -85,B 0,C 180,E1 -20854.748,E2 -20854.748} C_VEL
LIN {X 0,Y 214.381,Z 759.584,A -85,B 0,C 180,E1 -20857.852,E2 -20857.852} C_VEL
LIN {X 0,Y 215.104,Z 762.549,A -85,B 0,C 180,E1 -20861.345,E2 -20861.345} C_VEL
LIN {X 0,Y 216.482,Z 764.147,A -85,B 0,C 180,E1 -20864.947,E2 -20864.947} C_VEL
LIN {X 0,Y 217.488,Z 764.332,A -85,B 0,C 180,E1 -20866.926,E2 -20866.926} C_VEL
LIN {X 0,Y 218.721,Z 764.072,A -85,B 0,C 180,E1 -20868.884,E2 -20868.884} C_VEL
LIN {X 0,Y 220.443,Z 763.118,A -85,B 0,C 180,E1 -20871.218,E2 -20871.218} C_VEL
LIN {X 0,Y 223.431,Z 760.496,A -85,B 0,C 180,E1 -20874.585,E2 -20874.585} C_VEL
LIN {X 0,Y 226.618,Z 756.817,A -85,B 0,C 180,E1 -20877.473,E2 -20877.473} C_VEL
LIN {X 0,Y 230.417,Z 751.381,A -85,B 0,C 180,E1 -20880.481,E2 -20880.481} C_VEL
LIN {X 0,Y 234.21,Z 745.263,A -85,B 0,C 180,E1 -20883.01,E2 -20883.01} C_VEL
LIN {X 0,Y 235.646,Z 742.698,A -85,B 0,C 180,E1 -20883.89,E2 -20883.89} C_VEL
LIN {X 0,Y 236.982,Z 739.478,A -85,B 0,C 180,E1 -20885.047,E2 -20885.047} C_VEL
LIN {X 0,Y 237.716,Z 734.386,A -85,B 0,C 180,E1 -20887.096,E2 -20887.096} C_VEL
LIN {X 0,Y 238.495,Z 728.824,A -85,B 0,C 180,E1 -20889.044,E2 -20889.044} C_VEL
LIN {X 0,Y 239.831,Z 724.777,A -85,B 0,C 180,E1 -20890.021,E2 -20890.021} C_VEL
LIN {X 0,Y 243.387,Z 715.425,A -85,B 0,C 180,E1 -20891.662,E2 -20891.662} C_VEL
LIN {X 0,Y 247.221,Z 703.223,A -85,B 0,C 180,E1 -20893.381,E2 -20893.381} C_VEL
LIN {X 0,Y 250.127,Z 691.449,A -85,B 0,C 180,E1 -20894.648,E2 -20894.648} C_VEL
LIN {X 0,Y 252.463,Z 678.335,A -85,B 0,C 180,E1 -20895.749,E2 -20895.749} C_VEL
LIN {X 0,Y 254.025,Z 664.785,A -85,B 0,C 180,E1 -20896.553,E2 -20896.553} C_VEL
LIN {X 0,Y 257.024,Z 638.313,A -85,B 0,C 180,E1 -20897.826,E2 -20897.826} C_VEL
LIN {X 0,Y 253.801,Z 631.68,A -85,B 0,C 180,E1 -20900.154,E2 -20900.154} C_VEL
LIN {X 0,Y 250.558,Z 625.75,A -85,B 0,C 180,E1 -20903.044,E2 -20903.044} C_VEL
LIN {X 0,Y 249.028,Z 624.159,A -85,B 0,C 180,E1 -20904.565,E2 -20904.565} C_VEL
LIN {X 0,Y 247.081,Z 622.47,A -85,B 0,C 180,E1 -20907.072,E2 -20907.072} C_VEL
LIN {X 0,Y 245.207,Z 622.371,A -85,B 0,C 180,E1 -20911.058,E2 -20911.058} C_VEL
LIN {X 0,Y 244.901,Z 623.128,A -85,B 0,C 180,E1 -20913.253,E2 -20913.253} C_VEL
LIN {X 0,Y 245.366,Z 626.236,A -85,B 0,C 180,E1 -20916.729,E2 -20916.729} C_VEL
LIN {X 0,Y 246.798,Z 631.927,A -85,B 0,C 180,E1 -20920.083,E2 -20920.083} C_VEL
LIN {X 0,Y 248.262,Z 636.148,A -85,B 0,C 180,E1 -20922.155,E2 -20922.155} C_VEL
LIN {X 0,Y 250.294,Z 642.69,A -85,B 0,C 180,E1 -20924.468,E2 -20924.468} C_VEL
LIN {X 0,Y 252.21,Z 649.138,A -85,B 0,C 180,E1 -20926.273,E2 -20926.273} C_VEL
LIN {X 0,Y 252.55,Z 650.838,A -85,B 0,C 180,E1 -20926.634,E2 -20926.634} C_VEL
LIN {X 0,Y 252.475,Z 666.706,A -85,B 0,C 180,E1 -20928.218,E2 -20928.218} C_VEL
LIN {X 0,Y 251.977,Z 682.401,A -85,B 0,C 180,E1 -20929.467,E2 -20929.467} C_VEL
LIN {X 0,Y 251.139,Z 694.112,A -85,B 0,C 180,E1 -20930.186,E2 -20930.186} C_VEL
LIN {X 0,Y 248.641,Z 711.13,A -85,B 0,C 180,E1 -20930.936,E2 -20930.936} C_VEL
LIN {X 0,Y 245.288,Z 726.017,A -85,B 0,C 180,E1 -20931.846,E2 -20931.846} C_VEL
LIN {X 0,Y 241.068,Z 740.095,A -85,B 0,C 180,E1 -20933.04,E2 -20933.04} C_VEL
LIN {X 0,Y 236.747,Z 752.001,A -85,B 0,C 180,E1 -20934.37,E2 -20934.37} C_VEL
LIN {X 0,Y 232.127,Z 762.906,A -85,B 0,C 180,E1 -20935.939,E2 -20935.939} C_VEL
LIN {X 0,Y 226.437,Z 774.938,A -85,B 0,C 180,E1 -20938.157,E2 -20938.157} C_VEL
LIN {X 0,Y 222.924,Z 781.943,A -85,B 0,C 180,E1 -20939.775,E2 -20939.775} C_VEL
LIN {X 0,Y 220.683,Z 793.138,A -85,B 0,C 180,E1 -20941.207,E2 -20941.207} C_VEL
LIN {X 0,Y 217.855,Z 804.757,A -85,B 0,C 180,E1 -20943.153,E2 -20943.153} C_VEL
LIN {X 0,Y 214.944,Z 815.078,A -85,B 0,C 180,E1 -20945.364,E2 -20945.364} C_VEL
LIN {X 0,Y 212.129,Z 824.78,A -85,B 0,C 180,E1 -20948.073,E2 -20948.073} C_VEL
LIN {X 0,Y 209.622,Z 832.801,A -85,B 0,C 180,E1 -20950.922,E2 -20950.922} C_VEL
LIN {X 0,Y 207.946,Z 838.13,A -85,B 0,C 180,E1 -20953.307,E2 -20953.307} C_VEL
LIN {X 0,Y 206.337,Z 843.334,A -85,B 0,C 180,E1 -20956.208,E2 -20956.208} C_VEL
LIN {X 0,Y 205.331,Z 847.363,A -85,B 0,C 180,E1 -20959.151,E2 -20959.151} C_VEL
LIN {X 0,Y 204.671,Z 850.333,A -85,B 0,C 180,E1 -20962.107,E2 -20962.107} C_VEL
LIN {X 0,Y 204.439,Z 852.543,A -85,B 0,C 180,E1 -20965.515,E2 -20965.515} C_VEL
LIN {X 0,Y 204.456,Z 853.383,A -85,B 0,C 180,E1 -20968.032,E2 -20968.032} C_VEL
LIN {X 0,Y 204.568,Z 853.601,A -85,B 0,C 180,E1 -20970.002,E2 -20970.002} C_VEL
LIN {X 0,Y 204.449,Z 853.37,A -85,B 0,C 180,E1 -20971.972,E2 -20971.972} C_VEL
LIN {X 0,Y 204.439,Z 852.522,A -85,B 0,C 180,E1 -20974.489,E2 -20974.489} C_VEL
LIN {X 0,Y 204.677,Z 850.285,A -85,B 0,C 180,E1 -20977.896,E2 -20977.896} C_VEL
LIN {X 0,Y 205.329,Z 847.3,A -85,B 0,C 180,E1 -20980.852,E2 -20980.852} C_VEL
LIN {X 0,Y 206.305,Z 843.25,A -85,B 0,C 180,E1 -20983.797,E2 -20983.797} C_VEL
LIN {X 0,Y 208.256,Z 837.015,A -85,B 0,C 180,E1 -20987.176,E2 -20987.176} C_VEL
LIN {X 0,Y 210.42,Z 830.218,A -85,B 0,C 180,E1 -20990.021,E2 -20990.021} C_VEL
LIN {X 0,Y 212.872,Z 821.871,A -85,B 0,C 180,E1 -20992.776,E2 -20992.776} C_VEL
LIN {X 0,Y 215.41,Z 812.958,A -85,B 0,C 180,E1 -20995.097,E2 -20995.097} C_VEL
LIN {X 0,Y 218.073,Z 803.349,A -85,B 0,C 180,E1 -20997.08,E2 -20997.08} C_VEL
LIN {X 0,Y 220.682,Z 792.824,A -85,B 0,C 180,E1 -20998.797,E2 -20998.797} C_VEL
LIN {X 0,Y 223.011,Z 781.033,A -85,B 0,C 180,E1 -21000.281,E2 -21000.281} C_VEL
LIN {X 0,Y 225.045,Z 768.81,A -85,B 0,C 180,E1 -21001.41,E2 -21001.41} C_VEL
LIN {X 0,Y 226.716,Z 755.96,A -85,B 0,C 180,E1 -21002.211,E2 -21002.211} C_VEL
LIN {X 0,Y 227.632,Z 741.466,A -85,B 0,C 180,E1 -21002.765,E2 -21002.765} C_VEL
LIN {X 0,Y 229.737,Z 689.854,A -85,B 0,C 180,E1 -21004.313,E2 -21004.313} C_VEL
LIN {X 0,Y 227.723,Z 664.71,A -85,B 0,C 180,E1 -21005.604,E2 -21005.604} C_VEL
LIN {X 0,Y 224.667,Z 638.693,A -85,B 0,C 180,E1 -21007.173,E2 -21007.173} C_VEL
LIN {X 0,Y 224.005,Z 633.149,A -85,B 0,C 180,E1 -21007.58,E2 -21007.58} C_VEL
LIN {X 0,Y 224.466,Z 622.777,A -85,B 0,C 180,E1 -21009.026,E2 -21009.026} C_VEL
LIN {X 0,Y 221.756,Z 611.388,A -85,B 0,C 180,E1 -21011.323,E2 -21011.323} C_VEL
LIN {X 0,Y 218.816,Z 600.511,A -85,B 0,C 180,E1 -21013.731,E2 -21013.731} C_VEL
LIN {X 0,Y 216.829,Z 593.212,A -85,B 0,C 180,E1 -21015.487,E2 -21015.487} C_VEL
LIN {X 0,Y 211.999,Z 584.402,A -85,B 0,C 180,E1 -21018.469,E2 -21018.469} C_VEL
LIN {X 0,Y 209.92,Z 581.089,A -85,B 0,C 180,E1 -21019.873,E2 -21019.873} C_VEL
LIN {X 0,Y 209.39,Z 579.602,A -85,B 0,C 180,E1 -21020.378,E2 -21020.378} C_VEL
LIN {X 0,Y 207.316,Z 576.907,A -85,B 0,C 180,E1 -21021.754,E2 -21021.754} C_VEL
LIN {X 0,Y 206.693,Z 574.719,A -85,B 0,C 180,E1 -21022.57,E2 -21022.57} C_VEL
LIN {X 0,Y 206.702,Z 574.727,A -85,B 0,C 180,E1 -21027.043,E2 -21027.043} C_VEL
LIN {X 0,Y 206.77,Z 574.73,A -85,B 0,C 180,E1 -21032.097,E2 -21032.097} C_VEL
LIN {X 0,Y 206.757,Z 574.708,A -85,B 0,C 180,E1 -21036.605,E2 -21036.605} C_VEL
LIN {X 0,Y 206.875,Z 574.682,A -85,B 0,C 180,E1 -21042.197,E2 -21042.197} C_VEL
LIN {X 0,Y 206.896,Z 574.712,A -85,B 0,C 180,E1 -21046.244,E2 -21046.244} C_VEL
LIN {X 0,Y 207.103,Z 574.653,A -85,B 0,C 180,E1 -21050.231,E2 -21050.231} C_VEL
LIN {X 0,Y 207.064,Z 574.69,A -85,B 0,C 180,E1 -21054.156,E2 -21054.156} C_VEL
LIN {X 0,Y 207.384,Z 574.618,A -85,B 0,C 180,E1 -21058.058,E2 -21058.058} C_VEL
LIN {X 0,Y 207.514,Z 574.627,A -85,B 0,C 180,E1 -21060,E2 -21060} C_VEL
LIN {X 0,Y 207.384,Z 574.649,A -85,B 0,C 180,E1 -21061.942,E2 -21061.942} C_VEL
LIN {X 0,Y 207.17,Z 574.673,A -85,B 0,C 180,E1 -21067.799,E2 -21067.799} C_VEL
LIN {X 0,Y 206.946,Z 574.676,A -85,B 0,C 180,E1 -21071.757,E2 -21071.757} C_VEL
LIN {X 0,Y 206.871,Z 574.717,A -85,B 0,C 180,E1 -21075.771,E2 -21075.771} C_VEL
LIN {X 0,Y 206.787,Z 574.7,A -85,B 0,C 180,E1 -21079.869,E2 -21079.869} C_VEL
LIN {X 0,Y 206.767,Z 574.712,A -85,B 0,C 180,E1 -21084.072,E2 -21084.072} C_VEL
LIN {X 0,Y 206.748,Z 574.732,A -85,B 0,C 180,E1 -21088.418,E2 -21088.418} C_VEL
LIN {X 0,Y 206.728,Z 574.811,A -85,B 0,C 180,E1 -21092.225,E2 -21092.225} C_VEL
LIN {X 0,Y 207.081,Z 576.349,A -85,B 0,C 180,E1 -21092.889,E2 -21092.889} C_VEL
LIN {X 0,Y 209.968,Z 581.994,A -85,B 0,C 180,E1 -21095.897,E2 -21095.897} C_VEL
LIN {X 0,Y 213.421,Z 590.395,A -85,B 0,C 180,E1 -21099.729,E2 -21099.729} C_VEL
LIN {X 0,Y 216.376,Z 598.332,A -85,B 0,C 180,E1 -21103.008,E2 -21103.008} C_VEL
LIN {X 0,Y 219.667,Z 608.471,A -85,B 0,C 180,E1 -21106.708,E2 -21106.708} C_VEL
LIN {X 0,Y 222.351,Z 618.625,A -85,B 0,C 180,E1 -21110.023,E2 -21110.023} C_VEL
LIN {X 0,Y 224.263,Z 627.243,A -85,B 0,C 180,E1 -21112.48,E2 -21112.48} C_VEL
LIN {X 0,Y 226.652,Z 633.258,A -85,B 0,C 180,E1 -21113.179,E2 -21113.179} C_VEL
LIN {X 0,Y 230.706,Z 662.225,A -85,B 0,C 180,E1 -21115.022,E2 -21115.022} C_VEL
LIN {X 0,Y 231.221,Z 668.262,A -85,B 0,C 180,E1 -21115.336,E2 -21115.336} C_VEL
LIN {X 0,Y 227.965,Z 739.45,A -85,B 0,C 180,E1 -21117.479,E2 -21117.479} C_VEL
LIN {X 0,Y 226.724,Z 752.795,A -85,B 0,C 180,E1 -21118.198,E2 -21118.198} C_VEL
LIN {X 0,Y 224.98,Z 765.344,A -85,B 0,C 180,E1 -21119.233,E2 -21119.233} C_VEL
LIN {X 0,Y 223.004,Z 776.591,A -85,B 0,C 180,E1 -21120.499,E2 -21120.499} C_VEL
LIN {X 0,Y 220.694,Z 786.929,A -85,B 0,C 180,E1 -21121.983,E2 -21121.983} C_VEL
LIN {X 0,Y 218.023,Z 797.525,A -85,B 0,C 180,E1 -21123.946,E2 -21123.946} C_VEL
LIN {X 0,Y 215.52,Z 806.775,A -85,B 0,C 180,E1 -21126.12,E2 -21126.12} C_VEL
LIN {X 0,Y 212.904,Z 815.567,A -85,B 0,C 180,E1 -21128.707,E2 -21128.707} C_VEL
LIN {X 0,Y 210.389,Z 823.031,A -85,B 0,C 180,E1 -21131.496,E2 -21131.496} C_VEL
LIN {X 0,Y 208.396,Z 829.021,A -85,B 0,C 180,E1 -21134.347,E2 -21134.347} C_VEL
LIN {X 0,Y 206.826,Z 833.753,A -85,B 0,C 180,E1 -21137.238,E2 -21137.238} C_VEL
LIN {X 0,Y 205.715,Z 837.366,A -85,B 0,C 180,E1 -21140.163,E2 -21140.163} C_VEL
LIN {X 0,Y 205.198,Z 839.225,A -85,B 0,C 180,E1 -21142.124,E2 -21142.124} C_VEL
LIN {X 0,Y 204.764,Z 840.858,A -85,B 0,C 180,E1 -21144.476,E2 -21144.476} C_VEL
LIN {X 0,Y 204.49,Z 842.246,A -85,B 0,C 180,E1 -21148.029,E2 -21148.029} C_VEL
LIN {X 0,Y 204.497,Z 842.476,A -85,B 0,C 180,E1 -21149.998,E2 -21149.998} C_VEL
LIN {X 0,Y 204.471,Z 842.281,A -85,B 0,C 180,E1 -21151.968,E2 -21151.968} C_VEL
LIN {X 0,Y 204.822,Z 840.723,A -85,B 0,C 180,E1 -21155.907,E2 -21155.907} C_VEL
LIN {X 0,Y 205.194,Z 839.351,A -85,B 0,C 180,E1 -21157.873,E2 -21157.873} C_VEL
LIN {X 0,Y 206.022,Z 836.469,A -85,B 0,C 180,E1 -21160.812,E2 -21160.812} C_VEL
LIN {X 0,Y 207.259,Z 832.548,A -85,B 0,C 180,E1 -21163.729,E2 -21163.729} C_VEL
LIN {X 0,Y 208.937,Z 827.469,A -85,B 0,C 180,E1 -21166.612,E2 -21166.612} C_VEL
LIN {X 0,Y 211.094,Z 821.062,A -85,B 0,C 180,E1 -21169.445,E2 -21169.445} C_VEL
LIN {X 0,Y 213.78,Z 813.084,A -85,B 0,C 180,E1 -21172.212,E2 -21172.212} C_VEL
LIN {X 0,Y 216.295,Z 804.323,A -85,B 0,C 180,E1 -21174.643,E2 -21174.643} C_VEL
LIN {X 0,Y 218.825,Z 794.874,A -85,B 0,C 180,E1 -21176.718,E2 -21176.718} C_VEL
LIN {X 0,Y 221.279,Z 784.951,A -85,B 0,C 180,E1 -21178.449,E2 -21178.449} C_VEL
LIN {X 0,Y 223.535,Z 774.15,A -85,B 0,C 180,E1 -21179.939,E2 -21179.939} C_VEL
LIN {X 0,Y 225.588,Z 762.201,A -85,B 0,C 180,E1 -21181.192,E2 -21181.192} C_VEL
LIN {X 0,Y 227.147,Z 749.767,A -85,B 0,C 180,E1 -21182.124,E2 -21182.124} C_VEL
LIN {X 0,Y 228.201,Z 737.128,A -85,B 0,C 180,E1 -21182.741,E2 -21182.741} C_VEL
LIN {X 0,Y 231.167,Z 670.307,A -85,B 0,C 180,E1 -21184.743,E2 -21184.743} C_VEL
LIN {X 0,Y 228.536,Z 651.73,A -85,B 0,C 180,E1 -21185.908,E2 -21185.908} C_VEL
LIN {X 0,Y 225.053,Z 631.568,A -85,B 0,C 180,E1 -21187.345,E2 -21187.345} C_VEL
LIN {X 0,Y 223.283,Z 627.486,A -85,B 0,C 180,E1 -21187.88,E2 -21187.88} C_VEL
LIN {X 0,Y 222.088,Z 621.482,A -85,B 0,C 180,E1 -21189.808,E2 -21189.808} C_VEL
LIN {X 0,Y 220.284,Z 622.12,A -85,B 0,C 180,E1 -21190.03,E2 -21190.03} C_VEL
LIN {X 0,Y 217.723,Z 621.816,A -85,B 0,C 180,E1 -21190.69,E2 -21190.69} C_VEL
LIN {X 0,Y 217.105,Z 620.988,A -85,B 0,C 180,E1 -21191.065,E2 -21191.065} C_VEL
LIN {X 0,Y 215.983,Z 659.215,A -85,B 0,C 180,E1 -21192.883,E2 -21192.883} C_VEL
LIN {X 0,Y 215.315,Z 672.673,A -85,B 0,C 180,E1 -21193.872,E2 -21193.872} C_VEL
LIN {X 0,Y 214.387,Z 685.507,A -85,B 0,C 180,E1 -21195.185,E2 -21195.185} C_VEL
LIN {X 0,Y 213.255,Z 698.003,A -85,B 0,C 180,E1 -21196.856,E2 -21196.856} C_VEL
LIN {X 0,Y 211.947,Z 709.955,A -85,B 0,C 180,E1 -21198.888,E2 -21198.888} C_VEL
LIN {X 0,Y 210.634,Z 721.158,A -85,B 0,C 180,E1 -21201.273,E2 -21201.273} C_VEL
LIN {X 0,Y 209.539,Z 730.079,A -85,B 0,C 180,E1 -21203.603,E2 -21203.603} C_VEL
LIN {X 0,Y 208.324,Z 739.801,A -85,B 0,C 180,E1 -21206.756,E2 -21206.756} C_VEL
LIN {X 0,Y 207.696,Z 746.608,A -85,B 0,C 180,E1 -21209.498,E2 -21209.498} C_VEL
LIN {X 0,Y 207.345,Z 751.295,A -85,B 0,C 180,E1 -21211.792,E2 -21211.792} C_VEL
LIN {X 0,Y 207.09,Z 756.451,A -85,B 0,C 180,E1 -21214.899,E2 -21214.899} C_VEL
LIN {X 0,Y 207.347,Z 760.484,A -85,B 0,C 180,E1 -21218.109,E2 -21218.109} C_VEL
LIN {X 0,Y 207.984,Z 763.156,A -85,B 0,C 180,E1 -21221.104,E2 -21221.104} C_VEL
LIN {X 0,Y 209.163,Z 764.938,A -85,B 0,C 180,E1 -21224.407,E2 -21224.407} C_VEL
LIN {X 0,Y 210.149,Z 765.439,A -85,B 0,C 180,E1 -21226.461,E2 -21226.461} C_VEL
LIN {X 0,Y 211.388,Z 765.494,A -85,B 0,C 180,E1 -21228.493,E2 -21228.493} C_VEL
LIN {X 0,Y 213.338,Z 764.789,A -85,B 0,C 180,E1 -21231.206,E2 -21231.206} C_VEL
LIN {X 0,Y 216.163,Z 762.817,A -85,B 0,C 180,E1 -21234.402,E2 -21234.402} C_VEL
LIN {X 0,Y 219.294,Z 759.744,A -85,B 0,C 180,E1 -21237.314,E2 -21237.314} C_VEL
LIN {X 0,Y 222.644,Z 755.742,A -85,B 0,C 180,E1 -21240,E2 -21240} C_VEL
LIN {X 0,Y 226.502,Z 750.35,A -85,B 0,C 180,E1 -21242.668,E2 -21242.668} C_VEL
LIN {X 0,Y 230.774,Z 743.464,A -85,B 0,C 180,E1 -21245.242,E2 -21245.242} C_VEL
LIN {X 0,Y 235.056,Z 735.363,A -85,B 0,C 180,E1 -21247.634,E2 -21247.634} C_VEL
LIN {X 0,Y 239.199,Z 726.261,A -85,B 0,C 180,E1 -21249.726,E2 -21249.726} C_VEL
LIN {X 0,Y 239.831,Z 724.777,A -85,B 0,C 180,E1 -21250.021,E2 -21250.021} C_VEL
LIN {X 0,Y 241.206,Z 720.582,A -85,B 0,C 180,E1 -21250.961,E2 -21250.961} C_VEL
LIN {X 0,Y 242.167,Z 713.919,A -85,B 0,C 180,E1 -21252.692,E2 -21252.692} C_VEL
LIN {X 0,Y 242.972,Z 706.825,A -85,B 0,C 180,E1 -21254.301,E2 -21254.301} C_VEL
LIN {X 0,Y 244.029,Z 701.968,A -85,B 0,C 180,E1 -21255.038,E2 -21255.038} C_VEL
LIN {X 0,Y 247.119,Z 689.492,A -85,B 0,C 180,E1 -21256.31,E2 -21256.31} C_VEL
LIN {X 0,Y 249.249,Z 677.442,A -85,B 0,C 180,E1 -21257.269,E2 -21257.269} C_VEL
LIN {X 0,Y 251.619,Z 657.417,A -85,B 0,C 180,E1 -21258.391,E2 -21258.391} C_VEL
LIN {X 0,Y 253.428,Z 642.243,A -85,B 0,C 180,E1 -21259.132,E2 -21259.132} C_VEL
LIN {X 0,Y 250.935,Z 636.878,A -85,B 0,C 180,E1 -21261.195,E2 -21261.195} C_VEL
LIN {X 0,Y 248.371,Z 632.017,A -85,B 0,C 180,E1 -21263.744,E2 -21263.744} C_VEL
LIN {X 0,Y 246.555,Z 630.299,A -85,B 0,C 180,E1 -21265.772,E2 -21265.772} C_VEL
LIN {X 0,Y 245.519,Z 629.379,A -85,B 0,C 180,E1 -21267.258,E2 -21267.258} C_VEL
LIN {X 0,Y 243.757,Z 629.373,A -85,B 0,C 180,E1 -21271.264,E2 -21271.264} C_VEL
LIN {X 0,Y 243.479,Z 630.141,A -85,B 0,C 180,E1 -21273.26,E2 -21273.26} C_VEL
LIN {X 0,Y 243.779,Z 633.07,A -85,B 0,C 180,E1 -21276.396,E2 -21276.396} C_VEL
LIN {X 0,Y 245.141,Z 639.033,A -85,B 0,C 180,E1 -21279.896,E2 -21279.896} C_VEL
LIN {X 0,Y 246.199,Z 642.453,A -85,B 0,C 180,E1 -21281.541,E2 -21281.541} C_VEL
LIN {X 0,Y 247.934,Z 648.666,A -85,B 0,C 180,E1 -21283.751,E2 -21283.751} C_VEL
LIN {X 0,Y 249.435,Z 654.532,A -85,B 0,C 180,E1 -21285.417,E2 -21285.417} C_VEL
LIN {X 0,Y 249.12,Z 669.24,A -85,B 0,C 180,E1 -21286.913,E2 -21286.913} C_VEL
LIN {X 0,Y 248.343,Z 685.009,A -85,B 0,C 180,E1 -21288.182,E2 -21288.182} C_VEL
LIN {X 0,Y 247.535,Z 695.114,A -85,B 0,C 180,E1 -21288.8,E2 -21288.8} C_VEL
LIN {X 0,Y 245.094,Z 710.333,A -85,B 0,C 180,E1 -21289.486,E2 -21289.486} C_VEL
LIN {X 0,Y 241.667,Z 724.617,A -85,B 0,C 180,E1 -21290.362,E2 -21290.362} C_VEL
LIN {X 0,Y 237.245,Z 738.547,A -85,B 0,C 180,E1 -21291.534,E2 -21291.534} C_VEL
LIN {X 0,Y 232.182,Z 751.809,A -85,B 0,C 180,E1 -21293.018,E2 -21293.018} C_VEL
LIN {X 0,Y 226.879,Z 763.617,A -85,B 0,C 180,E1 -21294.767,E2 -21294.767} C_VEL
LIN {X 0,Y 221.473,Z 774.269,A -85,B 0,C 180,E1 -21296.814,E2 -21296.814} C_VEL
LIN {X 0,Y 216.572,Z 783.185,A -85,B 0,C 180,E1 -21298.994,E2 -21298.994} C_VEL
LIN {X 0,Y 214.116,Z 794.369,A -85,B 0,C 180,E1 -21300.507,E2 -21300.507} C_VEL
LIN {X 0,Y 211.188,Z 805.735,A -85,B 0,C 180,E1 -21302.503,E2 -21302.503} C_VEL
LIN {X 0,Y 208.507,Z 814.894,A -85,B 0,C 180,E1 -21304.55,E2 -21304.55} C_VEL
LIN {X 0,Y 205.947,Z 823.247,A -85,B 0,C 180,E1 -21306.897,E2 -21306.897} C_VEL
LIN {X 0,Y 203.332,Z 831.392,A -85,B 0,C 180,E1 -21309.781,E2 -21309.781} C_VEL
LIN {X 0,Y 201.129,Z 837.939,A -85,B 0,C 180,E1 -21312.724,E2 -21312.724} C_VEL
LIN {X 0,Y 199.406,Z 843.142,A -85,B 0,C 180,E1 -21315.719,E2 -21315.719} C_VEL
LIN {X 0,Y 198.318,Z 847.171,A -85,B 0,C 180,E1 -21318.762,E2 -21318.762} C_VEL
LIN {X 0,Y 197.637,Z 850.141,A -85,B 0,C 180,E1 -21321.824,E2 -21321.824} C_VEL
LIN {X 0,Y 197.337,Z 852.491,A -85,B 0,C 180,E1 -21325.71,E2 -21325.71} C_VEL
LIN {X 0,Y 197.358,Z 853.19,A -85,B 0,C 180,E1 -21327.961,E2 -21327.961} C_VEL
LIN {X 0,Y 197.483,Z 853.409,A -85,B 0,C 180,E1 -21330.002,E2 -21330.002} C_VEL
LIN {X 0,Y 197.351,Z 853.177,A -85,B 0,C 180,E1 -21332.042,E2 -21332.042} C_VEL
LIN {X 0,Y 197.338,Z 852.47,A -85,B 0,C 180,E1 -21334.293,E2 -21334.293} C_VEL
LIN {X 0,Y 197.643,Z 850.092,A -85,B 0,C 180,E1 -21338.179,E2 -21338.179} C_VEL
LIN {X 0,Y 198.312,Z 847.105,A -85,B 0,C 180,E1 -21341.241,E2 -21341.241} C_VEL
